C07288=1062.675,165.711,418.297,172.476,30.487,155.624
C07289=1062.681,165.960,418.274,172.478,30.490,155.624
C07290=1062.687,166.209,418.253,172.480,30.492,155.625
C07291=1062.693,166.458,418.230,172.483,30.496,155.625
C07292=1062.698,166.707,418.207,172.484,30.498,155.626
C07293=1062.704,166.956,418.185,172.486,30.501,155.626
C07294=1062.710,167.204,418.163,172.488,30.504,155.627
C07295=1062.715,167.454,418.140,172.490,30.507,155.627
C07296=1062.721,167.702,418.117,172.491,30.510,155.627
C07297=1062.727,167.952,418.096,172.494,30.513,155.628
C07298=1062.733,168.201,418.073,172.496,30.516,155.628
C07299=1062.738,168.449,418.050,172.498,30.519,155.629
C07300=1062.743,168.698,418.028,172.499,30.521,155.629
C07301=1062.750,168.947,418.006,172.501,30.524,155.630
C07302=1062.755,169.196,417.983,172.503,30.527,155.630
C07303=1062.761,169.445,417.960,172.506,30.530,155.631
C07304=1062.767,169.694,417.938,172.507,30.533,155.631
C07305=1062.773,169.943,417.916,172.509,30.536,155.632
C07306=1062.778,170.192,417.893,172.511,30.539,155.632
C07307=1062.784,170.440,417.870,172.513,30.541,155.632
C07308=1062.790,170.689,417.848,172.514,30.545,155.633
C07309=1062.795,170.939,417.826,172.517,30.547,155.633
C07310=1062.801,171.187,417.803,172.519,30.551,155.634
C07311=1062.807,171.436,417.780,172.521,30.553,155.634
C07312=1062.813,171.685,417.757,172.523,30.556,155.635
C07313=1062.819,171.934,417.735,172.524,30.559,155.635
C07314=1062.824,172.183,417.712,172.526,30.562,155.636
C07315=1062.830,172.431,417.690,172.529,30.565,155.636
C07316=1062.835,172.680,417.667,172.531,30.568,155.637
C07317=1062.842,172.930,417.645,172.532,30.571,155.637
C07318=1062.847,173.178,417.622,172.534,30.573,155.637
C07319=1062.853,173.427,417.599,172.536,30.576,155.638
C07320=1062.859,173.676,417.576,172.539,30.579,155.638
C07321=1062.865,173.925,417.554,172.540,30.582,155.639
C07322=1062.871,174.174,417.531,172.542,30.585,155.639
C07323=1062.877,174.458,417.506,172.545,30.589,155.640
C07324=1062.884,174.741,417.479,172.547,30.592,155.640
C07325=1062.891,175.024,417.453,172.549,30.595,155.641
C07326=1062.897,175.308,417.428,172.551,30.598,155.641
C07327=1062.903,175.557,417.405,172.553,30.601,155.642
C07328=1062.909,175.806,417.382,172.556,30.604,155.642
C07329=1062.914,176.055,417.359,172.557,30.607,155.643
C07330=1062.920,176.304,417.336,172.559,30.610,155.643
C07331=1062.927,176.552,417.314,172.561,30.612,155.644
C07332=1062.932,176.801,417.291,172.564,30.616,155.644
C07333=1062.938,177.050,417.268,172.565,30.618,155.645
C07334=1062.944,177.299,417.245,172.567,30.621,155.645
C07335=1062.950,177.548,417.222,172.569,30.624,155.646
C07336=1062.956,177.797,417.200,172.572,30.627,155.646
C07337=1062.962,178.045,417.177,172.573,30.630,155.646
C07338=1062.968,178.294,417.154,172.575,30.633,155.647
C07339=1062.974,178.544,417.131,172.577,30.636,155.647
C07340=1062.980,178.793,417.108,172.580,30.638,155.648
C07341=1062.985,179.042,417.085,172.581,30.642,155.648
C07342=1062.991,179.291,417.062,172.583,30.644,155.649
C07343=1062.997,179.539,417.039,172.585,30.647,155.649
C07344=1063.003,179.788,417.016,172.588,30.650,155.650
C07345=1063.009,180.037,416.993,172.590,30.653,155.650
C07346=1063.015,180.286,416.971,172.591,30.656,155.651
C07347=1063.020,180.535,416.948,172.593,30.659,155.651
C07348=1063.026,180.784,416.925,172.596,30.662,155.651
C07349=1063.033,181.033,416.901,172.598,30.665,155.652
C07350=1063.039,181.281,416.878,172.599,30.667,155.652
C07351=1063.045,181.530,416.855,172.601,30.670,155.653
C07352=1063.051,181.779,416.832,172.604,30.673,155.653
C07353=1063.056,182.028,416.809,172.606,30.676,155.654
C07354=1063.062,182.277,416.786,172.607,30.679,155.654
C07355=1063.068,182.526,416.764,172.610,30.682,155.655
C07356=1063.075,182.775,416.739,172.612,30.685,155.655
C07357=1063.080,183.024,416.717,172.614,30.687,155.655
C07358=1063.087,183.272,416.694,172.615,30.691,155.656
C07359=1063.092,183.521,416.671,172.618,30.693,155.656
C07360=1063.099,183.769,416.648,172.620,30.696,155.657
C07361=1063.105,184.019,416.624,172.622,30.699,155.657
C07362=1063.111,184.268,416.601,172.625,30.702,155.658
C07363=1063.116,184.517,416.578,172.626,30.705,155.658
C07364=1063.122,184.765,416.555,172.628,30.708,155.659
C07365=1063.127,185.014,416.531,172.631,30.711,155.659
C07366=1063.133,185.263,416.508,172.633,30.714,155.660
C07367=1063.139,185.511,416.485,172.634,30.717,155.660
C07368=1063.144,185.761,416.461,172.636,30.720,155.661
C07369=1063.150,186.010,416.438,172.639,30.723,155.661
C07370=1063.156,186.258,416.414,172.641,30.726,155.662
C07371=1063.161,186.508,416.391,172.642,30.730,155.662
C07372=1063.168,186.756,416.367,172.645,30.732,155.663
C07373=1063.172,187.005,416.343,172.647,30.736,155.663
C07374=1063.178,187.254,416.320,172.649,30.739,155.664
C07375=1063.184,187.502,416.297,172.650,30.742,155.664
C07376=1063.189,187.752,416.273,172.653,30.745,155.665
C07377=1063.195,188.000,416.250,172.655,30.748,155.665
C07378=1063.202,188.249,416.226,172.657,30.751,155.666
C07379=1063.207,188.498,416.202,172.659,30.754,155.666
C07380=1063.213,188.747,416.179,172.661,30.757,155.666
C07381=1063.218,188.996,416.155,172.663,30.760,155.667
C07382=1063.224,189.244,416.132,172.666,30.763,155.667
C07383=1063.230,189.493,416.108,172.668,30.766,155.668
C07384=1063.235,189.743,416.084,172.669,30.769,155.668
C07385=1063.241,189.991,416.061,172.672,30.773,155.669
C07386=1063.247,190.239,416.036,172.674,30.775,155.669
C07387=1063.253,190.523,416.010,172.677,30.779,155.670
C07388=1063.260,190.806,415.983,172.678,30.782,155.671
C07389=1063.267,191.089,415.957,172.681,30.786,155.671
C07390=1063.273,191.372,415.929,172.684,30.789,155.672
C07391=1063.279,191.620,415.906,172.686,30.792,155.672
C07392=1063.284,191.870,415.882,172.687,30.795,155.673
C07393=1063.290,192.118,415.858,172.690,30.798,155.673
C07394=1063.296,192.367,415.834,172.692,30.801,155.674
C07395=1063.301,192.616,415.811,172.694,30.805,155.674
C07396=1063.308,192.865,415.787,172.696,30.807,155.675
C07397=1063.313,193.114,415.762,172.698,30.811,155.675
C07398=1063.319,193.362,415.740,172.700,30.814,155.676
C07399=1063.325,193.612,415.715,172.703,30.817,155.676
C07400=1063.331,193.860,415.691,172.704,30.820,155.677
C07401=1063.336,194.109,415.668,172.707,30.823,155.677
C07402=1063.342,194.357,415.644,172.709,30.826,155.678
C07403=1063.348,194.607,415.619,172.711,30.829,155.678
C07404=1063.354,194.855,415.596,172.714,30.832,155.679
C07405=1063.359,195.104,415.572,172.715,30.835,155.679
C07406=1063.366,195.353,415.548,172.717,30.838,155.680
C07407=1063.372,195.601,415.525,172.720,30.842,155.680
C07408=1063.377,195.850,415.500,172.722,30.844,155.680
C07409=1063.384,196.099,415.476,172.724,30.848,155.681
C07410=1063.389,196.348,415.453,172.726,30.851,155.682
C07411=1063.395,196.597,415.429,172.728,30.853,155.682
C07412=1063.401,196.846,415.404,172.731,30.857,155.682
C07413=1063.407,197.094,415.381,172.732,30.860,155.683
C07414=1063.412,197.343,415.357,172.735,30.863,155.683
C07415=1063.419,197.592,415.332,172.737,30.866,155.684
C07416=1063.424,197.840,415.308,172.739,30.869,155.684
C07417=1063.430,198.089,415.284,172.742,30.872,155.685
C07418=1063.435,198.338,415.261,172.743,30.875,155.685
C07419=1063.441,198.587,415.237,172.746,30.879,155.686
C07420=1063.447,198.836,415.212,172.748,30.881,155.686
C07421=1063.453,199.084,415.189,172.751,30.884,155.687
C07422=1063.459,199.334,415.164,172.752,30.888,155.687
C07423=1063.465,199.582,415.140,172.754,30.891,155.688
C07424=1063.471,199.831,415.116,172.757,30.894,155.688
C07425=1063.477,200.079,415.092,172.759,30.897,155.689
C07426=1063.483,200.328,415.068,172.761,30.900,155.689
C07427=1063.489,200.577,415.044,172.763,30.903,155.690
C07428=1063.495,200.826,415.020,172.766,30.906,155.690
C07429=1063.500,201.075,414.995,172.768,30.909,155.691
C07430=1063.506,201.323,414.971,172.770,30.912,155.691
C07431=1063.512,201.572,414.947,172.772,30.915,155.692
C07432=1063.518,201.821,414.923,172.774,30.919,155.692
C07433=1063.524,202.070,414.898,172.777,30.921,155.693
C07434=1063.530,202.318,414.875,172.779,30.925,155.693
C07435=1063.537,202.567,414.849,172.781,30.928,155.694
C07436=1063.542,202.816,414.825,172.783,30.931,155.694
C07437=1063.548,203.065,414.801,172.786,30.934,155.695
C07438=1063.553,203.313,414.776,172.788,30.938,155.695
C07439=1063.559,203.562,414.753,172.790,30.941,155.696
C07440=1063.565,203.811,414.728,172.792,30.944,155.697
C07441=1063.571,204.059,414.703,172.794,30.947,155.697
C07442=1063.576,204.308,414.678,172.797,30.950,155.697
C07443=1063.582,204.557,414.654,172.799,30.953,155.698
C07444=1063.588,204.806,414.630,172.801,30.957,155.699
C07445=1063.594,205.054,414.606,172.803,30.960,155.699
C07446=1063.600,205.303,414.581,172.806,30.963,155.700
C07447=1063.605,205.552,414.556,172.808,30.966,155.700
C07448=1063.611,205.801,414.532,172.811,30.970,155.701
C07449=1063.617,206.049,414.507,172.812,30.973,155.701
C07450=1063.623,206.298,414.482,172.815,30.976,155.702
C07451=1063.647,207.346,414.379,172.981,31.057,155.708
C07452=1063.653,207.569,414.356,172.982,31.060,155.709
C07453=1063.659,207.793,414.333,172.984,31.064,155.710
C07454=1063.664,208.016,414.311,172.986,31.068,155.710
C07455=1063.669,208.240,414.288,172.988,31.071,155.711
C07456=1063.675,208.463,414.265,172.988,31.075,155.712
C07457=1063.680,208.688,414.242,172.990,31.079,155.712
C07458=1063.685,208.910,414.219,172.992,31.082,155.713
C07459=1063.691,209.134,414.196,172.994,31.086,155.714
C07460=1063.697,209.383,414.171,172.996,31.090,155.714
C07461=1063.703,209.631,414.146,172.998,31.094,155.715
C07462=1063.709,209.880,414.120,173.000,31.098,155.716
C07463=1063.715,210.129,414.094,173.002,31.102,155.717
C07464=1063.721,210.378,414.069,173.004,31.106,155.717
C07465=1063.728,210.626,414.043,173.006,31.111,155.718
C07466=1063.733,210.875,414.017,173.008,31.114,155.719
C07467=1063.739,211.123,413.992,173.010,31.119,155.720
C07468=1063.745,211.372,413.966,173.012,31.122,155.720
C07469=1063.752,211.621,413.941,173.014,31.127,155.721
C07470=1063.757,211.869,413.915,173.016,31.131,155.722
C07471=1063.763,212.117,413.889,173.018,31.135,155.722
C07472=1063.769,212.366,413.864,173.020,31.139,155.723
C07473=1063.775,212.615,413.838,173.022,31.143,155.724
C07474=1063.781,212.863,413.813,173.024,31.147,155.725
C07475=1063.787,213.112,413.787,173.026,31.151,155.725
C07476=1063.793,213.360,413.761,173.027,31.155,155.726
C07477=1063.799,213.609,413.735,173.030,31.159,155.727
C07478=1063.805,213.858,413.710,173.032,31.164,155.728
C07479=1063.811,214.106,413.683,173.034,31.167,155.728
C07480=1063.817,214.355,413.658,173.036,31.172,155.729
C07481=1063.823,214.604,413.632,173.037,31.175,155.730
C07482=1063.829,214.852,413.607,173.040,31.180,155.730
C07483=1063.835,215.101,413.580,173.042,31.184,155.731
C07484=1063.841,215.349,413.555,173.044,31.188,155.732
C07485=1063.847,215.598,413.528,173.045,31.192,155.733
C07486=1063.853,215.846,413.503,173.048,31.196,155.733
C07487=1063.858,216.095,413.477,173.050,31.200,155.734
C07488=1063.865,216.343,413.451,173.052,31.204,155.735
C07489=1063.871,216.592,413.426,173.054,31.208,155.736
C07490=1063.877,216.840,413.399,173.056,31.212,155.736
C07491=1063.884,217.090,413.373,173.058,31.216,155.737
C07492=1063.889,217.339,413.347,173.060,31.220,155.738
C07493=1063.896,217.587,413.321,173.062,31.225,155.738
C07494=1063.901,217.836,413.295,173.064,31.228,155.739
C07495=1063.908,218.084,413.269,173.066,31.233,155.740
C07496=1063.913,218.333,413.243,173.068,31.236,155.741
C07497=1063.920,218.581,413.217,173.070,31.240,155.741
C07498=1063.925,218.830,413.191,173.072,31.244,155.742
C07499=1063.932,219.078,413.165,173.074,31.248,155.743
C07500=1063.937,219.327,413.139,173.077,31.253,155.743
C07501=1063.944,219.576,413.113,173.079,31.256,155.744
C07502=1063.950,219.825,413.087,173.080,31.261,155.745
C07503=1063.956,220.073,413.061,173.083,31.264,155.746
C07504=1063.962,220.321,413.034,173.085,31.268,155.746
C07505=1063.968,220.570,413.009,173.087,31.272,155.747
C07506=1063.974,220.818,412.982,173.088,31.276,155.748
C07507=1063.980,221.067,412.957,173.091,31.281,155.748
C07508=1063.985,221.293,412.933,173.093,31.284,155.749
C07509=1063.991,221.519,412.909,173.095,31.287,155.750
C07510=1063.996,221.745,412.885,173.097,31.291,155.750
C07511=1064.002,221.971,412.861,173.098,31.295,155.751
C07512=1064.008,222.197,412.837,173.100,31.299,155.752
C07513=1064.013,222.423,412.813,173.102,31.302,155.752
C07514=1064.019,222.649,412.789,173.104,31.306,155.753
C07515=1064.023,222.875,412.765,173.106,31.310,155.754
C07516=1064.030,223.124,412.738,173.108,31.314,155.754
C07517=1064.036,223.372,412.712,173.110,31.318,155.755
C07518=1064.042,223.621,412.686,173.112,31.322,155.756
C07519=1064.047,223.869,412.660,173.115,31.326,155.757
C07520=1064.053,224.118,412.633,173.116,31.330,155.757
C07521=1064.060,224.366,412.607,173.118,31.334,155.758
C07522=1064.066,224.615,412.580,173.121,31.338,155.759
C07523=1064.072,224.864,412.554,173.123,31.342,155.759
C07524=1064.077,225.112,412.527,173.125,31.346,155.760
C07525=1064.084,225.360,412.501,173.127,31.350,155.761
C07526=1064.090,225.608,412.475,173.129,31.354,155.762
C07527=1064.096,225.857,412.448,173.131,31.358,155.762
C07528=1064.102,226.106,412.421,173.134,31.362,155.763
C07529=1064.107,226.355,412.395,173.135,31.366,155.764
C07530=1064.114,226.603,412.369,173.137,31.370,155.764
C07531=1064.120,226.852,412.342,173.140,31.374,155.765
C07532=1064.126,227.100,412.315,173.142,31.378,155.766
C07533=1064.132,227.349,412.289,173.145,31.382,155.767
C07534=1064.137,227.597,412.262,173.146,31.386,155.767
C07535=1064.145,227.846,412.236,173.148,31.390,155.768
C07536=1064.150,228.094,412.209,173.151,31.394,155.769
C07537=1064.156,228.342,412.182,173.153,31.398,155.769
C07538=1064.163,228.592,412.155,173.154,31.402,155.770
C07539=1064.168,228.840,412.129,173.157,31.406,155.771
C07540=1064.175,229.088,412.102,173.159,31.409,155.772
C07541=1064.181,229.337,412.075,173.161,31.414,155.772
C07542=1064.187,229.585,412.049,173.164,31.417,155.773
C07543=1064.193,229.834,412.022,173.165,31.422,155.774
C07544=1064.199,230.083,411.995,173.168,31.426,155.774
C07545=1064.205,230.331,411.969,173.170,31.429,155.775
C07546=1064.211,230.580,411.942,173.172,31.434,155.776
C07547=1064.216,230.828,411.915,173.175,31.437,155.777
C07548=1064.223,231.076,411.887,173.176,31.442,155.777
C07549=1064.229,231.325,411.861,173.179,31.445,155.778
C07550=1064.235,231.573,411.834,173.181,31.450,155.779
C07551=1064.241,231.822,411.807,173.183,31.453,155.779
C07552=1064.247,232.070,411.781,173.186,31.457,155.780
C07553=1064.253,232.319,411.754,173.187,31.462,155.781
C07554=1064.259,232.567,411.726,173.189,31.465,155.782
C07555=1064.265,232.816,411.700,173.192,31.470,155.782
C07556=1064.271,233.064,411.673,173.194,31.473,155.783
C07557=1064.277,233.313,411.646,173.197,31.477,155.784
C07558=1064.283,233.561,411.619,173.198,31.481,155.784
C07559=1064.289,233.810,411.591,173.200,31.485,155.785
C07560=1064.295,234.059,411.564,173.203,31.490,155.786
C07561=1064.300,234.307,411.538,173.205,31.493,155.787
C07562=1064.307,234.555,411.510,173.208,31.498,155.787
C07563=1064.313,234.804,411.483,173.209,31.501,155.788
C07564=1064.318,235.026,411.459,173.211,31.505,155.789
C07565=1064.323,235.248,411.435,173.213,31.508,155.789
C07566=1064.329,235.470,411.410,173.216,31.512,155.790
C07567=1064.334,235.691,411.386,173.218,31.516,155.791
C07568=1064.340,235.914,411.362,173.219,31.519,155.791
C07569=1064.345,236.136,411.337,173.221,31.523,155.792
C07570=1064.351,236.358,411.313,173.223,31.526,155.792
C07571=1064.356,236.580,411.289,173.225,31.530,155.793
C07572=1064.361,236.828,411.262,173.228,31.534,155.794
C07573=1064.368,237.077,411.235,173.230,31.538,155.795
C07574=1064.374,237.325,411.207,173.232,31.542,155.795
C07575=1064.380,237.574,411.180,173.234,31.545,155.796
C07576=1064.386,237.822,411.153,173.237,31.550,155.797
C07577=1064.392,238.071,411.126,173.239,31.554,155.797
C07578=1064.398,238.319,411.098,173.242,31.557,155.798
C07579=1064.404,238.568,411.071,173.243,31.562,155.799
C07580=1064.410,238.816,411.044,173.245,31.565,155.800
C07581=1064.416,239.065,411.016,173.248,31.569,155.800
C07582=1064.422,239.313,410.989,173.250,31.573,155.801
C07583=1064.429,239.562,410.962,173.253,31.577,155.802
C07584=1064.435,239.809,410.934,173.254,31.581,155.802
C07585=1064.441,240.058,410.906,173.257,31.585,155.803
C07586=1064.446,240.307,410.879,173.259,31.589,155.804
C07587=1064.453,240.555,410.852,173.262,31.593,155.805
C07588=1064.458,240.804,410.824,173.264,31.597,155.805
C07589=1064.465,241.052,410.797,173.267,31.601,155.806
C07590=1064.471,241.300,410.769,173.268,31.605,155.807
C07591=1064.477,241.549,410.742,173.271,31.609,155.807
C07592=1064.483,241.797,410.714,173.273,31.613,155.808
C07593=1064.489,242.045,410.687,173.276,31.617,155.809
C07594=1064.495,242.294,410.660,173.278,31.621,155.809
C07595=1064.501,242.542,410.632,173.280,31.625,155.810
C07596=1064.508,242.791,410.604,173.282,31.629,155.811
C07597=1064.513,243.040,410.577,173.284,31.632,155.812
C07598=1064.519,243.288,410.549,173.287,31.636,155.812
C07599=1064.525,243.536,410.521,173.289,31.641,155.813
C07600=1064.531,243.785,410.493,173.292,31.644,155.814
C07601=1064.537,244.033,410.465,173.293,31.649,155.815
C07602=1064.543,244.282,410.438,173.296,31.652,155.815
C07603=1064.548,244.530,410.410,173.298,31.657,155.816
C07604=1064.555,244.778,410.383,173.301,31.660,155.817
C07605=1064.560,245.026,410.355,173.303,31.664,155.817
C07606=1064.567,245.275,410.327,173.305,31.669,155.818
C07607=1064.573,245.523,410.299,173.307,31.672,155.819
C07608=1064.579,245.771,410.271,173.310,31.676,155.819
C07609=1064.585,246.021,410.244,173.312,31.680,155.820
C07610=1064.591,246.268,410.216,173.315,31.684,155.821
C07611=1064.597,246.517,410.188,173.317,31.688,155.822
C07612=1064.603,246.766,410.160,173.319,31.692,155.822
C07613=1064.609,247.013,410.132,173.322,31.696,155.823
C07614=1064.615,247.262,410.104,173.324,31.700,155.824
C07615=1064.620,247.510,410.076,173.327,31.704,155.824
C07616=1064.626,247.759,410.048,173.329,31.708,155.825
C07617=1064.633,248.007,410.020,173.332,31.712,155.826
C07618=1064.638,248.256,409.992,173.333,31.716,155.827
C07619=1064.644,248.504,409.964,173.336,31.720,155.827
C07620=1064.649,248.723,409.939,173.338,31.724,155.828
C07621=1064.654,248.942,409.914,173.340,31.727,155.829
C07622=1064.660,249.161,409.889,173.342,31.731,155.829
C07623=1064.665,249.380,409.864,173.345,31.734,155.830
C07624=1064.670,249.599,409.840,173.346,31.738,155.831
C07625=1064.675,249.818,409.815,173.348,31.741,155.831
C07626=1064.681,250.036,409.790,173.350,31.745,155.832
C07627=1064.686,250.255,409.765,173.352,31.748,155.833
C07628=1064.692,250.502,409.737,173.355,31.752,155.833
C07629=1064.698,250.751,409.709,173.358,31.757,155.834
C07630=1064.704,251.000,409.681,173.360,31.760,155.835
C07631=1064.709,251.248,409.653,173.362,31.764,155.835
C07632=1064.715,251.497,409.624,173.364,31.768,155.836
C07633=1064.722,251.745,409.597,173.367,31.772,155.837
C07634=1064.728,251.993,409.568,173.369,31.776,155.838
C07635=1064.734,252.241,409.540,173.372,31.780,155.838
C07636=1064.739,252.490,409.511,173.375,31.784,155.839
C07637=1064.745,252.739,409.483,173.376,31.788,155.840
C07638=1064.752,252.986,409.455,173.379,31.792,155.840
C07639=1064.758,253.235,409.427,173.381,31.796,155.841
C07640=1064.764,253.483,409.398,173.384,31.800,155.842
C07641=1064.770,253.732,409.369,173.386,31.804,155.843
C07642=1064.775,253.980,409.341,173.389,31.808,155.843
C07643=1064.782,254.228,409.313,173.391,31.812,155.844
C07644=1064.788,254.476,409.284,173.393,31.816,155.845
C07645=1064.794,254.725,409.256,173.396,31.820,155.845
C07646=1064.800,254.973,409.228,173.398,31.823,155.846
C07647=1064.806,255.221,409.199,173.401,31.828,155.847
C07648=1064.812,255.470,409.171,173.404,31.832,155.848
C07649=1064.819,255.718,409.142,173.406,31.835,155.848
C07650=1064.825,255.966,409.114,173.408,31.840,155.849
C07651=1064.830,256.214,409.085,173.410,31.843,155.850
C07652=1064.836,256.463,409.057,173.413,31.847,155.850
C07653=1064.842,256.711,409.029,173.416,31.851,155.851
C07654=1064.848,256.960,409.000,173.418,31.855,155.852
C07655=1064.854,257.208,408.971,173.421,31.859,155.853
C07656=1064.861,257.456,408.943,173.422,31.863,155.853
C07657=1064.867,257.705,408.915,173.425,31.867,155.854
C07658=1064.873,257.952,408.886,173.428,31.871,155.855
C07659=1064.879,258.200,408.857,173.430,31.875,155.855
C07660=1064.885,258.449,408.829,173.433,31.879,155.856
C07661=1064.891,258.697,408.799,173.436,31.883,155.857
C07662=1064.897,258.946,408.771,173.438,31.887,155.858
C07663=1064.904,259.194,408.742,173.440,31.891,155.858
C07664=1064.910,259.443,408.714,173.443,31.894,155.859
C07665=1064.917,259.691,408.685,173.445,31.898,155.860
C07666=1064.923,259.939,408.656,173.448,31.902,155.860
C07667=1064.929,260.188,408.628,173.450,31.906,155.861
C07668=1064.935,260.436,408.599,173.453,31.910,155.862
C07669=1064.941,260.684,408.570,173.456,31.914,155.863
C07670=1064.947,260.932,408.542,173.457,31.918,155.863
C07671=1064.953,261.180,408.513,173.460,31.922,155.864
C07672=1064.959,261.428,408.484,173.463,31.926,155.865
C07673=1064.965,261.676,408.455,173.465,31.929,155.865
C07674=1064.971,261.925,408.426,173.468,31.933,155.866
C07675=1064.977,262.173,408.397,173.471,31.938,155.867
C07676=1064.984,262.391,408.373,173.473,31.941,155.867
C07677=1064.989,262.609,408.347,173.475,31.944,155.868
C07678=1064.994,262.827,408.322,173.477,31.948,155.869
C07679=1065.000,263.045,408.296,173.479,31.951,155.869
C07680=1065.006,263.262,408.271,173.482,31.954,155.870
C07681=1065.011,263.480,408.246,173.484,31.958,155.871
C07682=1065.016,263.698,408.220,173.486,31.961,155.871
C07683=1065.022,263.915,408.194,173.489,31.965,155.872
C07684=1065.028,264.164,408.166,173.491,31.969,155.872
C07685=1065.033,264.412,408.136,173.493,31.973,155.873
C07686=1065.040,264.661,408.107,173.496,31.977,155.874
C07687=1065.045,264.908,408.079,173.498,31.981,155.875
C07688=1065.052,265.156,408.050,173.501,31.985,155.875
C07689=1065.057,265.405,408.020,173.504,31.989,155.876
C07690=1065.063,265.653,407.991,173.506,31.993,155.877
C07691=1065.070,265.901,407.962,173.509,31.996,155.878
C07692=1065.076,266.149,407.933,173.511,32.001,155.878
C07693=1065.081,266.397,407.903,173.514,32.005,155.879
C07694=1065.088,266.645,407.874,173.516,32.009,155.880
C07695=1065.094,266.894,407.845,173.519,32.012,155.880
C07696=1065.100,267.143,407.815,173.522,32.017,155.881
C07697=1065.106,267.391,407.786,173.524,32.020,155.882
C07698=1065.112,267.639,407.757,173.527,32.024,155.883
C07699=1065.119,267.887,407.727,173.530,32.029,155.883
C07700=1065.125,268.135,407.698,173.531,32.032,155.884
C07701=1065.131,268.383,407.669,173.534,32.037,155.885
C07702=1065.137,268.631,407.640,173.537,32.040,155.886
C07703=1065.143,268.880,407.610,173.540,32.044,155.886
C07704=1065.149,269.128,407.581,173.542,32.048,155.887
C07705=1065.155,269.376,407.552,173.545,32.052,155.888
C07706=1065.161,269.624,407.521,173.548,32.056,155.888
C07707=1065.167,269.872,407.492,173.551,32.060,155.889
C07708=1065.173,270.120,407.463,173.552,32.064,155.890
C07709=1065.179,270.369,407.433,173.555,32.068,155.891
C07710=1065.185,270.617,407.403,173.558,32.072,155.891
C07711=1065.192,270.865,407.374,173.561,32.076,155.892
C07712=1065.198,271.113,407.345,173.563,32.080,155.893
C07713=1065.203,271.362,407.315,173.566,32.084,155.894
C07714=1065.210,271.609,407.286,173.569,32.088,155.894
C07715=1065.215,271.858,407.256,173.572,32.092,155.895
C07716=1065.222,272.105,407.226,173.573,32.096,155.896
C07717=1065.228,272.354,407.196,173.576,32.100,155.897
C07718=1065.234,272.602,407.167,173.579,32.104,155.897
C07719=1065.240,272.850,407.137,173.582,32.108,155.898
C07720=1065.246,273.098,407.108,173.584,32.112,155.899
C07721=1065.252,273.347,407.078,173.587,32.116,155.899
C07722=1065.258,273.594,407.048,173.590,32.120,155.900
C07723=1065.264,273.843,407.019,173.593,32.124,155.901
C07724=1065.271,274.091,406.989,173.594,32.128,155.902
C07725=1065.277,274.339,406.959,173.597,32.132,155.902
C07726=1065.282,274.587,406.929,173.600,32.136,155.903
C07727=1065.289,274.835,406.900,173.603,32.140,155.904
C07728=1065.294,275.083,406.869,173.606,32.144,155.905
C07729=1065.301,275.332,406.840,173.608,32.148,155.905
C07730=1065.307,275.580,406.809,173.611,32.152,155.906
C07731=1065.313,275.828,406.779,173.614,32.156,155.907
C07732=1065.318,276.048,406.753,173.616,32.160,155.908
C07733=1065.323,276.267,406.727,173.618,32.163,155.908
C07734=1065.329,276.487,406.700,173.620,32.167,155.909
C07735=1065.335,276.706,406.674,173.623,32.170,155.909
C07736=1065.340,276.925,406.647,173.625,32.174,155.910
C07737=1065.346,277.145,406.621,173.628,32.178,155.911
C07738=1065.350,277.364,406.594,173.630,32.181,155.911
C07739=1065.356,277.584,406.567,173.633,32.185,155.912
C07740=1065.362,277.832,406.538,173.636,32.189,155.913
C07741=1065.368,278.080,406.507,173.638,32.192,155.914
C07742=1065.374,278.328,406.477,173.641,32.197,155.914
C07743=1065.380,278.577,406.447,173.643,32.201,155.915
C07744=1065.387,278.825,406.417,173.646,32.205,155.916
C07745=1065.393,279.073,406.387,173.649,32.209,155.916
C07746=1065.399,279.321,406.356,173.651,32.213,155.917
C07747=1065.405,279.569,406.327,173.654,32.217,155.918
C07748=1065.411,279.817,406.297,173.657,32.221,155.919
C07749=1065.417,280.066,406.266,173.660,32.225,155.920
C07750=1065.423,280.313,406.236,173.663,32.229,155.920
C07751=1065.429,280.561,406.205,173.666,32.233,155.921
C07752=1065.436,280.809,406.176,173.667,32.237,155.922
C07753=1065.442,281.058,406.146,173.670,32.241,155.923
C07754=1065.448,281.306,406.115,173.673,32.245,155.923
C07755=1065.453,281.553,406.085,173.676,32.249,155.924
C07756=1065.460,281.802,406.054,173.679,32.253,155.925
C07757=1065.466,282.050,406.024,173.682,32.258,155.926
C07758=1065.471,282.298,405.993,173.684,32.261,155.926
C07759=1065.478,282.546,405.963,173.687,32.266,155.927
C07760=1065.484,282.794,405.932,173.690,32.269,155.928
C07761=1065.489,283.042,405.902,173.693,32.274,155.929
C07762=1065.496,283.290,405.871,173.695,32.278,155.929
C07763=1065.502,283.538,405.841,173.698,32.282,155.930
C07764=1065.508,283.786,405.811,173.701,32.286,155.931
C07765=1065.514,284.034,405.780,173.704,32.290,155.932
C07766=1065.520,284.282,405.750,173.706,32.294,155.932
C07767=1065.526,284.531,405.719,173.709,32.298,155.933
C07768=1065.532,284.778,405.688,173.712,32.302,155.934
C07769=1065.539,285.026,405.658,173.715,32.306,155.935
C07770=1065.545,285.274,405.627,173.718,32.310,155.935
C07771=1065.551,285.522,405.597,173.721,32.314,155.936
C07772=1065.558,285.770,405.566,173.724,32.318,155.937
C07773=1065.563,286.018,405.536,173.726,32.323,155.938
C07774=1065.570,286.266,405.504,173.728,32.326,155.938
C07775=1065.576,286.514,405.474,173.731,32.331,155.939
C07776=1065.582,286.762,405.444,173.734,32.335,155.940
C07777=1065.588,287.010,405.413,173.737,32.339,155.941
C07778=1065.594,287.258,405.383,173.740,32.343,155.941
C07779=1065.601,287.506,405.351,173.743,32.347,155.942
C07780=1065.606,287.754,405.321,173.746,32.351,155.943
C07781=1065.613,288.002,405.290,173.749,32.355,155.944
C07782=1065.619,288.250,405.259,173.752,32.359,155.945
C07783=1065.625,288.498,405.228,173.755,32.363,155.945
C07784=1065.631,288.746,405.197,173.757,32.367,155.946
C07785=1065.637,288.994,405.166,173.760,32.372,155.947
C07786=1065.643,289.242,405.136,173.762,32.375,155.947
C07787=1065.649,289.490,405.105,173.765,32.380,155.948
C07788=1065.654,289.715,405.077,173.768,32.383,155.949
C07789=1065.661,289.940,405.049,173.771,32.387,155.950
C07790=1065.666,290.165,405.020,173.773,32.391,155.950
C07791=1065.672,290.389,404.993,173.776,32.394,155.951
C07792=1065.677,290.614,404.964,173.779,32.399,155.952
C07793=1065.683,290.839,404.936,173.781,32.402,155.953
C07794=1065.688,291.063,404.908,173.784,32.406,155.953
C07795=1065.694,291.288,404.879,173.787,32.410,155.954
C07796=1065.700,291.536,404.849,173.789,32.414,155.955
C07797=1065.706,291.784,404.818,173.792,32.418,155.955
C07798=1065.712,292.032,404.787,173.795,32.422,155.956
C07799=1065.718,292.280,404.755,173.798,32.426,155.957
C07800=1065.725,292.529,404.724,173.801,32.430,155.958
C07801=1065.731,292.776,404.693,173.803,32.435,155.959
C07802=1065.737,293.024,404.661,173.806,32.438,155.959
C07803=1065.743,293.272,404.631,173.809,32.443,155.960
C07804=1065.749,293.520,404.600,173.812,32.447,155.961
C07805=1065.755,293.768,404.568,173.815,32.451,155.962
C07806=1065.761,294.016,404.537,173.818,32.455,155.962
C07807=1065.768,294.264,404.506,173.821,32.459,155.963
C07808=1065.774,294.511,404.475,173.824,32.463,155.964
C07809=1065.780,294.760,404.443,173.827,32.468,155.965
C07810=1065.786,295.008,404.412,173.829,32.472,155.966
C07811=1065.792,295.255,404.380,173.832,32.476,155.966
C07812=1065.799,295.503,404.349,173.835,32.480,155.967
C07813=1065.805,295.752,404.318,173.838,32.484,155.968
C07814=1065.810,295.999,404.286,173.841,32.488,155.969
C07815=1065.817,296.247,404.255,173.844,32.493,155.969
C07816=1065.823,296.495,404.223,173.847,32.497,155.970
C07817=1065.829,296.742,404.192,173.850,32.501,155.971
C07818=1065.835,296.991,404.160,173.853,32.505,155.972
C07819=1065.842,297.239,404.129,173.856,32.510,155.973
C07820=1065.847,297.487,404.098,173.859,32.514,155.974
C07821=1065.854,297.735,404.066,173.862,32.518,155.974
C07822=1065.860,297.983,404.034,173.865,32.522,155.975
C07823=1065.865,298.230,404.002,173.868,32.527,155.976
C07824=1065.872,298.478,403.971,173.871,32.531,155.977
C07825=1065.878,298.726,403.939,173.873,32.535,155.978
C07826=1065.883,298.974,403.907,173.876,32.539,155.978
C07827=1065.889,299.222,403.875,173.879,32.544,155.979
C07828=1065.896,299.470,403.844,173.882,32.548,155.980
C07829=1065.902,299.717,403.811,173.885,32.552,155.981
C07830=1065.908,299.965,403.779,173.888,32.556,155.982
C07831=1065.914,300.213,403.748,173.891,32.561,155.982
C07832=1065.920,300.461,403.716,173.895,32.565,155.983
C07833=1065.926,300.709,403.684,173.898,32.569,155.984
C07834=1065.932,300.957,403.652,173.901,32.574,155.985
C07835=1065.938,301.205,403.621,173.904,32.578,155.986
C07836=1065.944,301.452,403.589,173.907,32.583,155.987
C07837=1065.950,301.700,403.556,173.910,32.587,155.987
C07838=1065.956,301.948,403.524,173.913,32.591,155.988
C07839=1065.963,302.196,403.493,173.916,32.595,155.989
C07840=1065.968,302.444,403.461,173.919,32.600,155.990
C07841=1065.974,302.691,403.429,173.922,32.604,155.991
C07842=1065.980,302.939,403.397,173.924,32.608,155.991
C07843=1065.987,303.187,403.365,173.927,32.612,155.992
C07844=1065.993,303.419,403.335,173.930,32.617,155.993
C07845=1065.998,303.651,403.305,173.933,32.620,155.994
C07846=1066.004,303.884,403.275,173.936,32.624,155.994
C07847=1066.010,304.116,403.245,173.939,32.629,155.995
C07848=1066.016,304.349,403.214,173.942,32.632,155.996
C07849=1066.021,304.581,403.185,173.945,32.637,155.997
C07850=1066.027,304.813,403.155,173.947,32.641,155.998
C07851=1066.033,305.045,403.125,173.950,32.644,155.998
C07852=1066.039,305.293,403.092,173.953,32.649,155.999
C07853=1066.045,305.541,403.060,173.957,32.654,156.000
C07854=1066.051,305.789,403.027,173.960,32.658,156.001
C07855=1066.058,306.037,402.996,173.963,32.662,156.002
C07856=1066.064,306.284,402.963,173.966,32.666,156.002
C07857=1066.070,306.533,402.931,173.969,32.670,156.003
C07858=1066.076,306.779,402.899,173.972,32.675,156.004
C07859=1066.082,307.028,402.867,173.975,32.679,156.005
C07860=1066.089,307.275,402.834,173.978,32.683,156.006
C07861=1066.095,307.523,402.802,173.982,32.688,156.007
C07862=1066.101,307.771,402.770,173.985,32.692,156.007
C07863=1066.107,308.019,402.738,173.988,32.697,156.008
C07864=1066.114,308.267,402.705,173.990,32.701,156.009
C07865=1066.120,308.514,402.672,173.993,32.705,156.010
C07866=1066.127,308.762,402.641,173.996,32.709,156.011
C07867=1066.133,309.010,402.608,173.999,32.713,156.011
C07868=1066.139,309.258,402.576,174.003,32.718,156.012
C07869=1066.145,309.505,402.543,174.006,32.723,156.013
C07870=1066.151,309.753,402.511,174.009,32.727,156.014
C07871=1066.158,310.001,402.478,174.012,32.731,156.015
C07872=1066.164,310.249,402.446,174.015,32.735,156.016
C07873=1066.170,310.496,402.413,174.018,32.740,156.017
C07874=1066.177,310.744,402.381,174.022,32.744,156.017
C07875=1066.184,310.992,402.348,174.025,32.749,156.018
C07876=1066.190,311.240,402.316,174.028,32.753,156.019
C07877=1066.196,311.488,402.283,174.031,32.757,156.020
C07878=1066.203,311.735,402.250,174.034,32.761,156.021
C07879=1066.209,311.983,402.217,174.038,32.766,156.022
C07880=1066.215,312.231,402.185,174.041,32.770,156.022
C07881=1066.221,312.479,402.153,174.044,32.775,156.023
C07882=1066.227,312.726,402.120,174.047,32.779,156.024
C07883=1066.234,312.975,402.087,174.050,32.783,156.025
C07884=1066.241,313.222,402.054,174.054,32.788,156.026
C07885=1066.247,313.470,402.021,174.057,32.792,156.027
C07886=1066.254,313.717,401.989,174.060,32.796,156.027
C07887=1066.260,313.965,401.956,174.063,32.800,156.028
C07888=1066.266,314.213,401.923,174.066,32.805,156.029
C07889=1066.272,314.460,401.890,174.070,32.810,156.030
C07890=1066.278,314.708,401.858,174.073,32.814,156.031
C07891=1066.284,314.956,401.824,174.076,32.819,156.032
C07892=1066.291,315.204,401.791,174.079,32.823,156.033
C07893=1066.296,315.452,401.758,174.082,32.828,156.034
C07894=1066.303,315.700,401.725,174.086,32.832,156.034
C07895=1066.309,315.947,401.692,174.089,32.837,156.035
C07896=1066.315,316.194,401.658,174.092,32.841,156.036
C07897=1066.321,316.442,401.626,174.095,32.846,156.037
C07898=1066.327,316.690,401.592,174.098,32.851,156.038
C07899=1066.333,316.938,401.560,174.102,32.855,156.039
C07900=1066.339,317.171,401.528,174.105,32.859,156.040
C07901=1066.345,317.406,401.496,174.108,32.864,156.041
C07902=1066.350,317.640,401.465,174.111,32.868,156.041
C07903=1066.357,317.874,401.433,174.114,32.872,156.042
C07904=1066.362,318.109,401.402,174.117,32.877,156.043
C07905=1066.368,318.342,401.371,174.120,32.881,156.044
C07906=1066.374,318.576,401.339,174.123,32.886,156.045
C07907=1066.380,318.811,401.307,174.126,32.890,156.046
C07908=1066.386,319.058,401.274,174.128,32.894,156.046
C07909=1066.392,319.306,401.241,174.132,32.899,156.047
C07910=1066.398,319.554,401.208,174.135,32.904,156.048
C07911=1066.405,319.802,401.174,174.138,32.908,156.049
C07912=1066.411,320.049,401.141,174.141,32.913,156.050
C07913=1066.417,320.297,401.107,174.145,32.917,156.051
C07914=1066.423,320.544,401.074,174.148,32.922,156.052
C07915=1066.429,320.793,401.040,174.151,32.926,156.053
C07916=1066.436,321.040,401.007,174.154,32.931,156.054
C07917=1066.441,321.288,400.973,174.158,32.935,156.054
C07918=1066.448,321.535,400.940,174.161,32.940,156.055
C07919=1066.454,321.783,400.906,174.164,32.945,156.056
C07920=1066.461,322.030,400.873,174.168,32.949,156.057
C07921=1066.467,322.279,400.839,174.171,32.954,156.058
C07922=1066.473,322.526,400.806,174.174,32.959,156.059
C07923=1066.479,322.773,400.772,174.177,32.963,156.060
C07924=1066.486,323.021,400.739,174.181,32.968,156.061
C07925=1066.492,323.269,400.704,174.185,32.972,156.062
C07926=1066.498,323.516,400.672,174.188,32.977,156.063
C07927=1066.505,323.764,400.637,174.192,32.982,156.064
C07928=1066.511,324.011,400.604,174.195,32.986,156.064
C07929=1066.518,324.260,400.570,174.198,32.991,156.065
C07930=1066.523,324.507,400.536,174.202,32.996,156.066
C07931=1066.531,324.755,400.502,174.205,33.000,156.067
C07932=1066.536,325.003,400.469,174.208,33.005,156.068
C07933=1066.543,325.250,400.435,174.212,33.009,156.069
C07934=1066.549,325.498,400.401,174.215,33.014,156.070
C07935=1066.556,325.745,400.368,174.218,33.019,156.071
C07936=1066.562,325.993,400.333,174.222,33.024,156.072
C07937=1066.568,326.240,400.300,174.225,33.028,156.073
C07938=1066.575,326.488,400.266,174.228,33.033,156.074
C07939=1066.581,326.736,400.232,174.232,33.037,156.075
C07940=1066.588,326.983,400.198,174.235,33.042,156.075
C07941=1066.595,327.231,400.164,174.238,33.047,156.076
C07942=1066.600,327.478,400.130,174.242,33.052,156.077
C07943=1066.608,327.726,400.096,174.245,33.056,156.078
C07944=1066.613,327.974,400.062,174.249,33.061,156.079
C07945=1066.620,328.222,400.029,174.252,33.065,156.080
C07946=1066.626,328.469,399.995,174.255,33.070,156.081
C07947=1066.633,328.717,399.960,174.259,33.075,156.082
C07948=1066.640,328.965,399.926,174.262,33.080,156.083
C07949=1066.646,329.212,399.892,174.266,33.085,156.084
C07950=1066.652,329.460,399.858,174.269,33.089,156.085
C07951=1066.659,329.707,399.824,174.272,33.094,156.086
C07952=1066.665,329.955,399.790,174.276,33.099,156.087
C07953=1066.672,330.202,399.755,174.279,33.103,156.088
C07954=1066.679,330.449,399.721,174.283,33.108,156.089
C07955=1066.685,330.697,399.687,174.286,33.113,156.089
C07956=1066.691,330.929,399.656,174.289,33.117,156.090
C07957=1066.697,331.160,399.623,174.292,33.122,156.091
C07958=1066.703,331.391,399.591,174.296,33.126,156.092
C07959=1066.708,331.621,399.559,174.299,33.131,156.093
C07960=1066.715,331.853,399.527,174.302,33.136,156.094
C07961=1066.721,332.084,399.495,174.305,33.140,156.095
C07962=1066.726,332.315,399.462,174.308,33.144,156.096
C07963=1066.732,332.547,399.430,174.312,33.149,156.097
C07964=1066.738,332.794,399.396,174.315,33.154,156.098
C07965=1066.745,333.041,399.361,174.318,33.159,156.099
C07966=1066.751,333.289,399.326,174.323,33.164,156.100
C07967=1066.757,333.536,399.292,174.326,33.169,156.101
C07968=1066.764,333.784,399.257,174.330,33.173,156.102
C07969=1066.771,334.032,399.223,174.333,33.178,156.102
C07970=1066.776,334.279,399.189,174.337,33.184,156.104
C07971=1066.783,334.526,399.153,174.340,33.188,156.104
C07972=1066.790,334.774,399.119,174.344,33.193,156.105
C07973=1066.796,335.022,399.084,174.347,33.198,156.106
C07974=1066.802,335.269,399.050,174.351,33.203,156.107
C07975=1066.809,335.516,399.015,174.354,33.208,156.108
C07976=1066.816,335.764,398.980,174.358,33.213,156.109
C07977=1066.822,336.012,398.945,174.361,33.218,156.110
C07978=1066.828,336.259,398.911,174.365,33.223,156.111
C07979=1066.835,336.506,398.876,174.368,33.228,156.112
C07980=1066.842,336.754,398.841,174.371,33.232,156.113
C07981=1066.848,337.002,398.806,174.375,33.238,156.114
C07982=1066.855,337.249,398.771,174.379,33.243,156.115
C07983=1066.860,337.497,398.737,174.382,33.248,156.116
C07984=1066.867,337.744,398.701,174.385,33.253,156.117
C07985=1066.874,337.991,398.666,174.390,33.258,156.118
C07986=1066.880,338.239,398.632,174.394,33.263,156.119
C07987=1066.886,338.487,398.596,174.397,33.268,156.121
C07988=1066.892,338.734,398.561,174.401,33.273,156.121
C07989=1066.899,338.981,398.526,174.404,33.278,156.123
C07990=1066.906,339.229,398.491,174.408,33.283,156.124
C07991=1066.911,339.477,398.456,174.411,33.288,156.125
C07992=1066.918,339.724,398.421,174.415,33.293,156.126
C07993=1066.925,339.972,398.386,174.418,33.298,156.127
C07994=1066.930,340.219,398.351,174.422,33.303,156.128
C07995=1066.937,340.466,398.315,174.425,33.308,156.129
C07996=1066.944,340.713,398.280,174.429,33.313,156.130
C07997=1066.950,340.961,398.245,174.432,33.318,156.131
C07998=1066.957,341.208,398.209,174.436,33.324,156.132
C07999=1066.964,341.456,398.174,174.440,33.329,156.133
C08000=1066.969,341.704,398.139,174.444,33.334,156.134
C08001=1066.976,341.951,398.104,174.448,33.339,156.135
C08002=1066.983,342.199,398.069,174.451,33.344,156.136
C08003=1066.989,342.446,398.033,174.455,33.349,156.137
C08004=1066.996,342.693,397.997,174.458,33.354,156.138
C08005=1067.003,342.940,397.962,174.462,33.360,156.139
C08006=1067.009,343.188,397.927,174.465,33.365,156.140
C08007=1067.015,343.436,397.891,174.469,33.370,156.141
C08008=1067.022,343.683,397.856,174.473,33.375,156.142
C08009=1067.028,343.931,397.821,174.476,33.380,156.143
C08010=1067.035,344.178,397.785,174.481,33.385,156.144
C08011=1067.041,344.426,397.750,174.484,33.391,156.145
C08012=1067.047,344.654,397.717,174.488,33.395,156.146
C08013=1067.052,344.882,397.684,174.491,33.401,156.147
C08014=1067.059,345.111,397.651,174.494,33.405,156.148
C08015=1067.065,345.339,397.618,174.498,33.410,156.149
C08016=1067.071,345.569,397.585,174.501,33.415,156.150
C08017=1067.077,345.797,397.552,174.504,33.420,156.151
C08018=1067.083,346.026,397.518,174.508,33.425,156.152
C08019=1067.089,346.254,397.486,174.511,33.430,156.153
C08020=1067.095,346.502,397.450,174.515,33.435,156.155
C08021=1067.102,346.749,397.414,174.519,33.440,156.156
C08022=1067.108,346.996,397.378,174.523,33.446,156.157
C08023=1067.114,347.243,397.342,174.527,33.451,156.158
C08024=1067.121,347.491,397.307,174.530,33.456,156.159
C08025=1067.128,347.739,397.271,174.534,33.461,156.160
C08026=1067.135,347.986,397.235,174.538,33.467,156.161
C08027=1067.141,348.234,397.199,174.541,33.472,156.162
C08028=1067.147,348.481,397.163,174.545,33.478,156.163
C08029=1067.154,348.728,397.126,174.549,33.483,156.164
C08030=1067.160,348.975,397.091,174.553,33.488,156.165
C08031=1067.167,349.222,397.055,174.557,33.494,156.167
C08032=1067.173,349.470,397.019,174.561,33.499,156.168
C08033=1067.180,349.717,396.983,174.564,33.504,156.169
C08034=1067.187,349.964,396.946,174.568,33.510,156.170
C08035=1067.193,350.212,396.911,174.572,33.516,156.171
C08036=1067.200,350.459,396.875,174.575,33.521,156.172
C08037=1067.206,350.706,396.838,174.579,33.526,156.173
C08038=1067.213,350.954,396.802,174.584,33.532,156.174
C08039=1067.219,351.201,396.766,174.588,33.537,156.176
C08040=1067.226,351.448,396.730,174.591,33.542,156.177
C08041=1067.233,351.695,396.693,174.595,33.548,156.178
C08042=1067.239,351.943,396.657,174.599,33.553,156.179
C08043=1067.245,352.190,396.621,174.602,33.559,156.180
C08044=1067.252,352.438,396.585,174.606,33.564,156.181
C08045=1067.259,352.684,396.549,174.611,33.570,156.182
C08046=1067.265,352.931,396.512,174.615,33.575,156.183
C08047=1067.272,353.179,396.475,174.618,33.581,156.185
C08048=1067.279,353.426,396.439,174.622,33.586,156.186
C08049=1067.285,353.673,396.403,174.626,33.592,156.187
C08050=1067.292,353.921,396.366,174.630,33.598,156.188
C08051=1067.298,354.168,396.329,174.633,33.603,156.189
C08052=1067.304,354.415,396.293,174.638,33.609,156.190
C08053=1067.311,354.662,396.256,174.642,33.615,156.192
C08054=1067.318,354.910,396.220,174.646,33.620,156.193
C08055=1067.324,355.157,396.183,174.649,33.626,156.194
C08056=1067.330,355.404,396.147,174.653,33.632,156.195
C08057=1067.337,355.652,396.110,174.657,33.637,156.196
C08058=1067.344,355.899,396.073,174.661,33.643,156.197
C08059=1067.350,356.146,396.037,174.665,33.648,156.199
C08060=1067.357,356.393,395.999,174.669,33.654,156.200
C08061=1067.364,356.640,395.963,174.673,33.660,156.201
C08062=1067.371,356.888,395.926,174.677,33.666,156.202
C08063=1067.377,357.135,395.890,174.681,33.671,156.203
C08064=1067.384,357.381,395.853,174.684,33.677,156.205
C08065=1067.390,357.629,395.816,174.689,33.682,156.206
C08066=1067.397,357.876,395.779,174.693,33.688,156.207
C08067=1067.404,358.123,395.742,174.697,33.694,156.208
C08068=1067.414,358.502,395.686,174.703,33.703,156.210
C08069=1067.425,358.881,395.629,174.710,33.711,156.212
C08070=1067.434,359.260,395.573,174.716,33.721,156.214
C08071=1067.445,359.638,395.515,174.721,33.729,156.216
C08072=1067.451,359.885,395.479,174.725,33.735,156.217
C08073=1067.458,360.133,395.441,174.729,33.741,156.218
C08074=1067.465,360.380,395.405,174.734,33.747,156.219
C08075=1067.471,360.627,395.367,174.738,33.753,156.221
C08076=1067.478,360.874,395.330,174.742,33.759,156.222
C08077=1067.485,361.121,395.293,174.746,33.764,156.223
C08078=1067.491,361.368,395.256,174.749,33.770,156.224
C08079=1067.498,361.616,395.218,174.754,33.776,156.226
C08080=1067.504,361.862,395.181,174.758,33.782,156.227
C08081=1067.511,362.110,395.144,174.762,33.788,156.228
C08082=1067.518,362.356,395.107,174.766,33.794,156.229
C08083=1067.524,362.604,395.069,174.770,33.800,156.231
C08084=1067.532,362.851,395.031,174.775,33.806,156.232
C08085=1067.538,363.098,394.995,174.779,33.811,156.233
C08086=1067.545,363.345,394.957,174.783,33.818,156.234
C08087=1067.551,363.592,394.920,174.786,33.823,156.236
C08088=1067.558,363.839,394.882,174.791,33.830,156.237
C08089=1067.566,364.086,394.844,174.795,33.835,156.238
C08090=1067.572,364.333,394.807,174.799,33.842,156.239
C08091=1067.579,364.581,394.770,174.803,33.847,156.241
C08092=1067.588,364.910,394.720,174.808,33.855,156.242
C08093=1067.596,365.239,394.669,174.815,33.864,156.244
C08094=1067.605,365.569,394.619,174.820,33.872,156.246
C08095=1067.614,365.899,394.568,174.825,33.880,156.248
C08096=1067.621,366.146,394.531,174.830,33.886,156.249
C08097=1067.627,366.392,394.493,174.834,33.893,156.250
C08098=1067.634,366.639,394.455,174.838,33.898,156.252
C08099=1067.641,366.886,394.417,174.842,33.905,156.253
C08100=1067.648,367.133,394.380,174.847,33.911,156.254
C08101=1067.654,367.380,394.341,174.851,33.917,156.256
C08102=1067.661,367.627,394.304,174.855,33.923,156.257
C08103=1067.668,367.875,394.266,174.859,33.929,156.258
C08104=1067.674,368.121,394.227,174.864,33.935,156.260
C08105=1067.681,368.368,394.190,174.868,33.942,156.261
C08106=1067.688,368.616,394.152,174.872,33.948,156.262
C08107=1067.695,368.862,394.113,174.876,33.954,156.264
C08108=1067.701,369.109,394.076,174.881,33.961,156.265
C08109=1067.708,369.356,394.038,174.885,33.967,156.266
C08110=1067.715,369.603,393.999,174.889,33.973,156.268
C08111=1067.722,369.850,393.961,174.893,33.979,156.269
C08112=1067.729,370.097,393.924,174.898,33.986,156.270
C08113=1067.736,370.344,393.885,174.902,33.992,156.272
C08114=1067.742,370.591,393.848,174.906,33.998,156.273
C08115=1067.749,370.837,393.809,174.911,34.004,156.274
C08116=1067.756,371.085,393.771,174.915,34.011,156.276
C08117=1067.763,371.331,393.732,174.919,34.017,156.277
C08118=1067.770,371.579,393.694,174.923,34.024,156.279
C08119=1067.777,371.826,393.656,174.928,34.030,156.280
C08120=1067.784,372.065,393.619,174.932,34.036,156.281
C08121=1067.790,372.304,393.581,174.936,34.042,156.283
C08122=1067.797,372.544,393.544,174.940,34.049,156.284
C08123=1067.804,372.783,393.507,174.945,34.055,156.285
C08124=1067.811,373.022,393.470,174.949,34.061,156.287
C08125=1067.817,373.261,393.433,174.953,34.067,156.288
C08126=1067.823,373.500,393.395,174.958,34.074,156.289
C08127=1067.830,373.740,393.358,174.962,34.080,156.291
C08128=1067.836,373.986,393.319,174.966,34.087,156.292
C08129=1067.843,374.233,393.281,174.971,34.093,156.294
C08130=1067.850,374.480,393.242,174.975,34.100,156.295
C08131=1067.857,374.727,393.203,174.979,34.106,156.297
C08132=1067.864,374.974,393.164,174.983,34.113,156.298
C08133=1067.871,375.220,393.126,174.988,34.119,156.299
C08134=1067.878,375.467,393.087,174.992,34.126,156.301
C08135=1067.885,375.714,393.048,174.996,34.133,156.302
C08136=1067.892,375.961,393.009,175.002,34.139,156.304
C08137=1067.899,376.208,392.970,175.006,34.146,156.305
C08138=1067.905,376.454,392.932,175.010,34.153,156.307
C08139=1067.912,376.701,392.893,175.015,34.160,156.308
C08140=1067.919,376.948,392.854,175.019,34.166,156.310
C08141=1067.926,377.195,392.815,175.023,34.173,156.311
C08142=1067.933,377.442,392.776,175.028,34.179,156.312
C08143=1067.939,377.688,392.737,175.033,34.186,156.314
C08144=1067.947,377.936,392.698,175.037,34.193,156.315
C08145=1067.954,378.182,392.659,175.042,34.200,156.317
C08146=1067.961,378.429,392.620,175.046,34.206,156.318
C08147=1067.968,378.676,392.581,175.051,34.213,156.320
C08148=1067.974,378.923,392.542,175.055,34.220,156.321
C08149=1067.981,379.169,392.503,175.060,34.227,156.323
C08150=1067.988,379.416,392.464,175.065,34.234,156.324
C08151=1067.996,379.663,392.425,175.069,34.241,156.326
C08152=1068.003,379.909,392.385,175.073,34.247,156.327
C08153=1068.010,380.156,392.346,175.079,34.254,156.329
C08154=1068.017,380.402,392.307,175.083,34.261,156.330
C08155=1068.024,380.650,392.267,175.087,34.268,156.332
C08156=1068.031,380.897,392.229,175.092,34.275,156.334
C08157=1068.038,381.143,392.189,175.096,34.282,156.335
C08158=1068.045,381.390,392.150,175.102,34.289,156.337
C08159=1068.052,381.637,392.110,175.106,34.296,156.338
C08160=1068.059,381.883,392.070,175.110,34.303,156.340
C08161=1068.066,382.130,392.031,175.115,34.310,156.341
C08162=1068.072,382.377,391.991,175.120,34.317,156.343
C08163=1068.080,382.624,391.952,175.125,34.324,156.344
C08164=1068.087,382.870,391.912,175.129,34.331,156.346
C08165=1068.093,383.117,391.872,175.133,34.338,156.348
C08166=1068.100,383.363,391.833,175.139,34.345,156.349
C08167=1068.108,383.611,391.793,175.143,34.352,156.351
C08168=1068.114,383.857,391.753,175.148,34.360,156.352
C08169=1068.121,384.103,391.714,175.153,34.367,156.354
C08170=1068.129,384.350,391.674,175.158,34.374,156.356
C08171=1068.135,384.597,391.634,175.162,34.381,156.357
C08172=1068.142,384.843,391.594,175.166,34.388,156.359
C08173=1068.149,385.090,391.554,175.172,34.395,156.360
C08174=1068.156,385.336,391.514,175.176,34.403,156.362
C08175=1068.164,385.584,391.475,175.181,34.410,156.364
C08176=1068.171,385.845,391.432,175.186,34.418,156.365
C08177=1068.178,386.107,391.390,175.192,34.425,156.367
C08178=1068.187,386.369,391.347,175.196,34.433,156.369
C08179=1068.193,386.631,391.305,175.202,34.441,156.371
C08180=1068.201,386.877,391.265,175.206,34.448,156.372
C08181=1068.208,387.124,391.225,175.211,34.456,156.374
C08182=1068.215,387.371,391.185,175.216,34.463,156.375
C08183=1068.222,387.616,391.144,175.220,34.470,156.377
C08184=1068.229,387.864,391.104,175.226,34.478,156.379
C08185=1068.237,388.110,391.064,175.230,34.485,156.380
C08186=1068.244,388.357,391.024,175.236,34.492,156.382
C08187=1068.251,388.603,390.984,175.240,34.500,156.384
C08188=1068.259,388.850,390.944,175.245,34.507,156.385
C08189=1068.265,389.096,390.904,175.250,34.515,156.387
C08190=1068.273,389.342,390.863,175.255,34.522,156.389
C08191=1068.280,389.590,390.822,175.260,34.530,156.390
C08192=1068.287,389.836,390.783,175.265,34.537,156.392
C08193=1068.295,390.082,390.742,175.270,34.545,156.394
C08194=1068.302,390.329,390.702,175.275,34.552,156.396
C08195=1068.309,390.575,390.661,175.280,34.560,156.397
C08196=1068.317,390.822,390.621,175.285,34.567,156.399
C08197=1068.323,391.068,390.580,175.289,34.575,156.401
C08198=1068.330,391.315,390.540,175.295,34.583,156.402
C08199=1068.338,391.561,390.499,175.299,34.591,156.404
C08200=1068.345,391.807,390.458,175.305,34.598,156.406
C08201=1068.352,392.055,390.418,175.309,34.605,156.408
C08202=1068.360,392.301,390.377,175.315,34.613,156.409
C08203=1068.367,392.547,390.336,175.319,34.621,156.411
C08204=1068.374,392.794,390.296,175.325,34.629,156.413
C08205=1068.381,393.041,390.254,175.330,34.637,156.415
C08206=1068.388,393.286,390.214,175.335,34.645,156.417
C08207=1068.396,393.533,390.173,175.340,34.652,156.418
C08208=1068.403,393.779,390.132,175.345,34.660,156.420
C08209=1068.410,394.027,390.091,175.350,34.668,156.422
C08210=1068.417,394.273,390.050,175.355,34.676,156.424
C08211=1068.425,394.519,390.010,175.360,34.684,156.426
C08212=1068.432,394.765,389.968,175.365,34.692,156.427
C08213=1068.439,395.012,389.927,175.371,34.700,156.429
C08214=1068.447,395.259,389.886,175.376,34.708,156.431
C08215=1068.454,395.505,389.845,175.381,34.716,156.433
C08216=1068.461,395.751,389.804,175.386,34.724,156.435
C08217=1068.468,395.998,389.763,175.391,34.732,156.437
C08218=1068.475,396.244,389.721,175.396,34.740,156.438
C08219=1068.483,396.490,389.679,175.402,34.748,156.440
C08220=1068.490,396.737,389.638,175.407,34.756,156.442
C08221=1068.497,396.983,389.597,175.412,34.764,156.444
C08222=1068.505,397.230,389.556,175.417,34.772,156.446
C08223=1068.513,397.476,389.515,175.422,34.780,156.448
C08224=1068.520,397.722,389.473,175.428,34.789,156.450
C08225=1068.527,397.969,389.432,175.433,34.797,156.451
C08226=1068.535,398.215,389.391,175.438,34.805,156.453
C08227=1068.542,398.462,389.348,175.444,34.813,156.455
C08228=1068.549,398.708,389.307,175.449,34.822,156.457
C08229=1068.556,398.954,389.265,175.454,34.830,156.459
C08230=1068.564,399.201,389.224,175.460,34.838,156.461
C08231=1068.571,399.447,389.182,175.464,34.846,156.463
C08232=1068.579,399.725,389.135,175.471,34.856,156.465
C08233=1068.588,400.003,389.088,175.477,34.865,156.467
C08234=1068.596,400.281,389.041,175.483,34.875,156.469
C08235=1068.605,400.558,388.994,175.489,34.884,156.472
C08236=1068.612,400.804,388.952,175.494,34.893,156.474
C08237=1068.619,401.051,388.910,175.500,34.901,156.476
C08238=1068.626,401.297,388.868,175.505,34.910,156.478
C08239=1068.635,401.544,388.826,175.510,34.918,156.480
C08240=1068.642,401.790,388.784,175.516,34.927,156.482
C08241=1068.650,402.037,388.743,175.522,34.935,156.483
C08242=1068.656,402.283,388.700,175.527,34.944,156.485
C08243=1068.664,402.529,388.658,175.532,34.952,156.488
C08244=1068.672,402.775,388.616,175.538,34.961,156.489
C08245=1068.680,403.021,388.574,175.543,34.969,156.491
C08246=1068.687,403.268,388.532,175.549,34.978,156.494
C08247=1068.694,403.514,388.490,175.554,34.987,156.496
C08248=1068.702,403.761,388.448,175.560,34.995,156.498
C08249=1068.709,404.007,388.406,175.565,35.004,156.500
C08250=1068.717,404.253,388.364,175.571,35.013,156.502
C08251=1068.725,404.499,388.321,175.577,35.022,156.504
C08252=1068.732,404.746,388.278,175.582,35.031,156.506
C08253=1068.739,404.992,388.236,175.587,35.039,156.508
C08254=1068.747,405.239,388.193,175.593,35.048,156.510
C08255=1068.755,405.485,388.151,175.599,35.057,156.512
C08256=1068.761,405.731,388.109,175.605,35.066,156.514
C08257=1068.770,405.977,388.066,175.611,35.075,156.516
C08258=1068.777,406.223,388.023,175.616,35.084,156.518
C08259=1068.785,406.470,387.981,175.621,35.093,156.521
C08260=1068.792,406.716,387.938,175.627,35.102,156.523
C08261=1068.800,406.962,387.895,175.633,35.111,156.525
C08262=1068.807,407.208,387.853,175.639,35.120,156.527
C08263=1068.814,407.454,387.809,175.645,35.129,156.529
C08264=1068.823,407.701,387.767,175.650,35.138,156.531
C08265=1068.830,407.946,387.724,175.656,35.148,156.533
C08266=1068.837,408.193,387.681,175.662,35.157,156.536
C08267=1068.845,408.439,387.638,175.668,35.166,156.538
C08268=1068.853,408.686,387.595,175.674,35.175,156.540
C08269=1068.860,408.931,387.552,175.680,35.184,156.542
C08270=1068.868,409.178,387.509,175.686,35.194,156.544
C08271=1068.876,409.425,387.466,175.691,35.203,156.547
C08272=1068.883,409.670,387.423,175.697,35.212,156.549
C08273=1068.891,409.916,387.380,175.703,35.222,156.551
C08274=1068.898,410.162,387.337,175.709,35.231,156.553
C08275=1068.906,410.409,387.294,175.715,35.240,156.555
C08276=1068.914,410.655,387.251,175.721,35.250,156.558
C08277=1068.922,410.901,387.207,175.727,35.259,156.560
C08278=1068.929,411.147,387.164,175.733,35.269,156.562
C08279=1068.937,411.393,387.120,175.739,35.278,156.564
C08280=1068.945,411.639,387.078,175.745,35.288,156.567
C08281=1068.953,411.885,387.034,175.751,35.297,156.569
C08282=1068.961,412.131,386.990,175.757,35.306,156.571
C08283=1068.968,412.378,386.947,175.763,35.316,156.574
C08284=1068.976,412.623,386.904,175.769,35.326,156.576
C08285=1068.984,412.869,386.860,175.776,35.335,156.578
C08286=1068.992,413.116,386.817,175.781,35.345,156.581
C08287=1068.999,413.362,386.773,175.787,35.355,156.583
C08288=1069.008,413.644,386.723,175.795,35.366,156.586
C08289=1069.018,413.926,386.673,175.802,35.377,156.588
C08290=1069.027,414.208,386.623,175.809,35.388,156.591
C08291=1069.036,414.489,386.573,175.816,35.399,156.594
C08292=1069.044,414.735,386.530,175.822,35.409,156.596
C08293=1069.052,414.981,386.486,175.828,35.419,156.598
C08294=1069.060,415.227,386.442,175.834,35.429,156.601
C08295=1069.067,415.473,386.397,175.840,35.439,156.603
C08296=1069.075,415.720,386.354,175.847,35.449,156.606
C08297=1069.083,415.965,386.309,175.853,35.459,156.608
C08298=1069.091,416.211,386.265,175.859,35.469,156.611
C08299=1069.099,416.458,386.221,175.866,35.479,156.613
C08300=1069.107,416.703,386.177,175.873,35.489,156.615
C08301=1069.115,416.949,386.133,175.879,35.499,156.618
C08302=1069.123,417.195,386.089,175.885,35.509,156.620
C08303=1069.131,417.441,386.045,175.892,35.519,156.623
C08304=1069.139,417.687,386.000,175.898,35.530,156.625
C08305=1069.147,417.933,385.956,175.904,35.540,156.628
C08306=1069.154,418.179,385.911,175.911,35.550,156.630
C08307=1069.162,418.424,385.867,175.917,35.561,156.633
C08308=1069.170,418.671,385.823,175.924,35.571,156.635
C08309=1069.178,418.917,385.779,175.931,35.581,156.638
C08310=1069.186,419.162,385.735,175.937,35.592,156.640
C08311=1069.194,419.408,385.690,175.943,35.602,156.643
C08312=1069.203,419.654,385.645,175.950,35.612,156.645
C08313=1069.211,419.900,385.600,175.956,35.623,156.648
C08314=1069.219,420.146,385.556,175.964,35.634,156.651
C08315=1069.227,420.391,385.511,175.970,35.644,156.653
C08316=1069.235,420.637,385.467,175.977,35.654,156.656
C08317=1069.244,420.884,385.422,175.983,35.665,156.658
C08318=1069.251,421.129,385.377,175.991,35.676,156.661
C08319=1069.259,421.375,385.332,175.997,35.686,156.664
C08320=1069.268,421.621,385.288,176.004,35.697,156.666
C08321=1069.276,421.867,385.242,176.010,35.708,156.669
C08322=1069.284,422.112,385.198,176.018,35.719,156.672
C08323=1069.291,422.358,385.152,176.024,35.729,156.674
C08324=1069.300,422.604,385.107,176.031,35.740,156.677
C08325=1069.308,422.850,385.062,176.037,35.751,156.680
C08326=1069.316,423.095,385.017,176.045,35.762,156.682
C08327=1069.325,423.341,384.972,176.051,35.773,156.685
C08328=1069.332,423.587,384.926,176.058,35.784,156.688
C08329=1069.340,423.832,384.882,176.066,35.795,156.690
C08330=1069.349,424.079,384.836,176.072,35.806,156.693
C08331=1069.357,424.324,384.791,176.079,35.817,156.696
C08332=1069.365,424.570,384.745,176.086,35.828,156.699
C08333=1069.374,424.815,384.700,176.093,35.840,156.702
C08334=1069.382,425.062,384.654,176.101,35.851,156.704
C08335=1069.390,425.307,384.609,176.107,35.862,156.707
C08336=1069.398,425.553,384.563,176.114,35.873,156.710
C08337=1069.407,425.798,384.518,176.122,35.884,156.713
C08338=1069.415,426.044,384.472,176.129,35.896,156.715
C08339=1069.423,426.289,384.427,176.136,35.907,156.718
C08340=1069.431,426.536,384.381,176.143,35.918,156.721
C08341=1069.441,426.781,384.335,176.151,35.929,156.724
C08342=1069.448,427.026,384.289,176.158,35.941,156.727
C08343=1069.457,427.272,384.244,176.165,35.952,156.730
C08344=1069.468,427.573,384.187,176.173,35.966,156.733
C08345=1069.478,427.874,384.131,176.182,35.980,156.737
C08346=1069.488,428.175,384.075,176.192,35.995,156.740
C08347=1069.498,428.475,384.018,176.201,36.009,156.744
C08348=1069.506,428.721,383.972,176.208,36.021,156.747
C08349=1069.515,428.966,383.926,176.215,36.032,156.750
C08350=1069.523,429.213,383.880,176.223,36.044,156.753
C08351=1069.532,429.458,383.834,176.230,36.056,156.756
C08352=1069.540,429.703,383.788,176.238,36.068,156.759
C08353=1069.548,429.949,383.741,176.245,36.080,156.762
C08354=1069.557,430.194,383.694,176.253,36.092,156.765
C08355=1069.565,430.440,383.648,176.261,36.103,156.768
C08356=1069.574,430.686,383.602,176.268,36.115,156.771
C08357=1069.583,430.931,383.556,176.276,36.127,156.774
C08358=1069.591,431.176,383.509,176.283,36.139,156.777
C08359=1069.599,431.421,383.463,176.291,36.151,156.780
C08360=1069.608,431.667,383.416,176.299,36.163,156.783
C08361=1069.616,431.912,383.369,176.307,36.176,156.786
C08362=1069.625,432.158,383.322,176.314,36.188,156.789
C08363=1069.634,432.403,383.276,176.322,36.201,156.792
C08364=1069.642,432.649,383.229,176.330,36.213,156.796
C08365=1069.651,432.894,383.182,176.337,36.225,156.799
C08366=1069.659,433.139,383.135,176.345,36.238,156.802
C08367=1069.668,433.385,383.088,176.353,36.250,156.805
C08368=1069.677,433.630,383.041,176.361,36.262,156.808
C08369=1069.685,433.875,382.994,176.369,36.275,156.811
C08370=1069.694,434.121,382.947,176.376,36.287,156.815
C08371=1069.703,434.366,382.900,176.385,36.300,156.818
C08372=1069.711,434.612,382.852,176.393,36.313,156.821
C08373=1069.719,434.857,382.806,176.401,36.325,156.824
C08374=1069.728,435.102,382.758,176.409,36.338,156.828
C08375=1069.737,435.347,382.711,176.417,36.351,156.831
C08376=1069.746,435.593,382.664,176.425,36.363,156.834
C08377=1069.755,435.838,382.616,176.433,36.376,156.838
C08378=1069.764,436.083,382.569,176.441,36.389,156.841
C08379=1069.772,436.328,382.522,176.449,36.402,156.844
C08380=1069.781,436.574,382.474,176.458,36.415,156.848
C08381=1069.790,436.819,382.426,176.466,36.428,156.851
C08382=1069.799,437.064,382.379,176.474,36.441,156.854
C08383=1069.808,437.309,382.331,176.483,36.454,156.858
C08384=1069.817,437.554,382.283,176.491,36.467,156.861
C08385=1069.826,437.799,382.236,176.499,36.480,156.864
C08386=1069.835,438.045,382.188,176.508,36.493,156.868
C08387=1069.843,438.290,382.140,176.516,36.506,156.871
C08388=1069.852,438.535,382.093,176.525,36.519,156.875
C08389=1069.862,438.781,382.045,176.533,36.533,156.878
C08390=1069.870,439.025,381.996,176.541,36.546,156.882
C08391=1069.880,439.271,381.948,176.550,36.559,156.885
C08392=1069.888,439.516,381.901,176.559,36.573,156.889
C08393=1069.897,439.761,381.852,176.568,36.587,156.892
C08394=1069.906,440.006,381.804,176.576,36.600,156.896
C08395=1069.915,440.251,381.755,176.585,36.613,156.899
C08396=1069.924,440.496,381.708,176.593,36.627,156.903
C08397=1069.934,440.741,381.659,176.602,36.641,156.907
C08398=1069.942,440.986,381.611,176.611,36.655,156.910
C08399=1069.952,441.231,381.563,176.620,36.668,156.914
C08400=1069.959,441.446,381.520,176.628,36.680,156.917
C08401=1069.967,441.661,381.478,176.636,36.693,156.920
C08402=1069.975,441.875,381.435,176.643,36.705,156.923
C08403=1069.984,442.090,381.392,176.651,36.717,156.927
C08404=1069.992,442.305,381.350,176.659,36.729,156.930
C08405=1069.999,442.520,381.307,176.667,36.741,156.933
C08406=1070.007,442.734,381.264,176.675,36.754,156.936
C08407=1070.016,442.949,381.221,176.683,36.766,156.940
C08408=1070.024,443.193,381.173,176.691,36.780,156.943
C08409=1070.034,443.438,381.124,176.701,36.794,156.947
C08410=1070.043,443.684,381.075,176.710,36.808,156.951
C08411=1070.052,443.929,381.026,176.720,36.823,156.955
C08412=1070.062,444.173,380.977,176.728,36.837,156.959
C08413=1070.071,444.418,380.928,176.738,36.851,156.962
C08414=1070.080,444.663,380.879,176.747,36.866,156.966
C08415=1070.090,444.908,380.830,176.757,36.881,156.970
C08416=1070.099,445.153,380.780,176.766,36.895,156.974
C08417=1070.108,445.397,380.731,176.776,36.910,156.978
C08418=1070.117,445.643,380.681,176.784,36.924,156.982
C08419=1070.127,445.887,380.632,176.794,36.939,156.986
C08420=1070.136,446.132,380.582,176.803,36.954,156.990
C08421=1070.145,446.377,380.533,176.813,36.968,156.994
C08422=1070.155,446.622,380.483,176.823,36.983,156.998
C08423=1070.164,446.866,380.434,176.832,36.998,157.002
C08424=1070.174,447.111,380.384,176.842,37.013,157.006
C08425=1070.183,447.355,380.335,176.852,37.028,157.010
C08426=1070.192,447.601,380.285,176.861,37.043,157.014
C08427=1070.202,447.846,380.235,176.871,37.058,157.018
C08428=1070.212,448.089,380.186,176.881,37.073,157.022
C08429=1070.222,448.332,380.136,176.891,37.088,157.026
C08430=1070.233,448.577,380.087,176.899,37.102,157.030
C08431=1070.245,448.822,380.039,176.908,37.117,157.034
C08432=1070.259,449.066,379.992,176.916,37.130,157.037
C08433=1070.273,449.311,379.945,176.925,37.143,157.041
C08434=1070.289,449.556,379.899,176.933,37.156,157.044
C08435=1070.306,449.802,379.854,176.940,37.168,157.048
C08436=1069.957,449.802,379.601,176.927,37.307,157.085
C08437=1069.941,449.557,379.646,176.920,37.295,157.081
C08438=1069.925,449.312,379.692,176.911,37.282,157.078
C08439=1069.911,449.067,379.739,176.903,37.269,157.074
C08440=1069.897,448.822,379.786,176.894,37.255,157.071
C08441=1069.885,448.577,379.835,176.886,37.241,157.067
C08442=1069.873,448.332,379.884,176.876,37.227,157.063
C08443=1069.863,448.088,379.932,176.866,37.212,157.059
C08444=1069.853,447.845,379.982,176.856,37.197,157.055
C08445=1069.843,447.601,380.032,176.847,37.182,157.051
C08446=1069.834,447.356,380.082,176.837,37.167,157.047
C08447=1069.825,447.111,380.131,176.827,37.152,157.043
C08448=1069.815,446.867,380.181,176.817,37.137,157.039
C08449=1069.806,446.622,380.231,176.807,37.122,157.035
C08450=1069.795,446.377,380.281,176.798,37.108,157.031
C08451=1069.786,446.132,380.330,176.788,37.093,157.027
C08452=1069.777,445.887,380.380,176.778,37.078,157.023
C08453=1069.768,445.642,380.429,176.769,37.063,157.019
C08454=1069.758,445.398,380.479,176.759,37.049,157.015
C08455=1069.749,445.153,380.528,176.749,37.034,157.011
C08456=1069.739,444.908,380.578,176.741,37.020,157.007
C08457=1069.730,444.663,380.627,176.731,37.005,157.003
C08458=1069.721,444.419,380.676,176.722,36.991,156.999
C08459=1069.712,444.174,380.725,176.712,36.977,156.995
C08460=1069.703,443.929,380.775,176.703,36.962,156.991
C08461=1069.693,443.684,380.823,176.693,36.948,156.988
C08462=1069.684,443.439,380.872,176.685,36.934,156.984
C08463=1069.675,443.194,380.921,176.675,36.920,156.980
C08464=1069.665,442.949,380.970,176.666,36.905,156.976
C08465=1069.650,442.539,381.052,176.651,36.882,156.970
C08466=1069.634,442.127,381.133,176.636,36.859,156.964
C08467=1069.619,441.717,381.215,176.621,36.835,156.958
C08468=1069.603,441.307,381.296,176.606,36.812,156.952
C08469=1069.594,441.062,381.345,176.596,36.798,156.948
C08470=1069.585,440.817,381.393,176.587,36.785,156.944
C08471=1069.577,440.572,381.442,176.579,36.771,156.941
C08472=1069.567,440.327,381.490,176.569,36.758,156.937
C08473=1069.558,440.082,381.539,176.561,36.744,156.933
C08474=1069.549,439.836,381.587,176.552,36.730,156.930
C08475=1069.541,439.592,381.636,176.544,36.717,156.926
C08476=1069.531,439.346,381.683,176.535,36.704,156.923
C08477=1069.522,439.101,381.731,176.526,36.690,156.919
C08478=1069.513,438.856,381.780,176.517,36.677,156.916
C08479=1069.504,438.611,381.827,176.509,36.663,156.912
C08480=1069.496,438.366,381.875,176.500,36.650,156.909
C08481=1069.486,438.121,381.924,176.492,36.637,156.905
C08482=1069.478,437.876,381.971,176.484,36.624,156.902
C08483=1069.468,437.630,382.019,176.475,36.611,156.899
C08484=1069.459,437.386,382.067,176.467,36.598,156.895
C08485=1069.450,437.140,382.114,176.457,36.585,156.892
C08486=1069.441,436.895,382.162,176.449,36.572,156.888
C08487=1069.433,436.650,382.210,176.441,36.559,156.885
C08488=1069.423,436.404,382.258,176.433,36.546,156.882
C08489=1069.415,436.159,382.304,176.424,36.533,156.878
C08490=1069.406,435.914,382.352,176.416,36.520,156.875
C08491=1069.397,435.669,382.399,176.408,36.508,156.872
C08492=1069.388,435.423,382.447,176.399,36.495,156.868
C08493=1069.379,435.178,382.494,176.391,36.482,156.865
C08494=1069.370,434.933,382.541,176.384,36.469,156.862
C08495=1069.362,434.688,382.589,176.376,36.457,156.858
C08496=1069.354,434.442,382.636,176.368,36.444,156.855
C08497=1069.345,434.197,382.684,176.359,36.432,156.852
C08498=1069.336,433.951,382.731,176.351,36.419,156.849
C08499=1069.327,433.706,382.778,176.343,36.407,156.846
C08500=1069.318,433.461,382.825,176.335,36.394,156.842
C08501=1069.310,433.215,382.872,176.327,36.382,156.839
C08502=1069.301,432.970,382.919,176.319,36.369,156.836
C08503=1069.292,432.725,382.966,176.312,36.357,156.833
C08504=1069.284,432.479,383.012,176.304,36.345,156.830
C08505=1069.275,432.234,383.059,176.296,36.332,156.826
C08506=1069.267,431.988,383.106,176.288,36.320,156.823
C08507=1069.258,431.743,383.153,176.281,36.308,156.820
C08508=1069.250,431.499,383.200,176.273,36.296,156.817
C08509=1069.241,431.253,383.246,176.265,36.284,156.814
C08510=1069.233,431.007,383.292,176.257,36.272,156.811
C08511=1069.225,430.761,383.339,176.250,36.260,156.808
C08512=1069.216,430.516,383.386,176.242,36.248,156.805
C08513=1069.208,430.270,383.433,176.234,36.236,156.802
C08514=1069.198,430.025,383.479,176.227,36.224,156.799
C08515=1069.190,429.779,383.525,176.219,36.212,156.796
C08516=1069.181,429.534,383.572,176.211,36.200,156.793
C08517=1069.173,429.289,383.618,176.204,36.188,156.790
C08518=1069.165,429.043,383.663,176.196,36.177,156.787
C08519=1069.156,428.797,383.710,176.188,36.165,156.784
C08520=1069.147,428.552,383.757,176.182,36.154,156.781
C08521=1069.138,428.250,383.814,176.172,36.139,156.777
C08522=1069.126,427.947,383.870,176.163,36.125,156.774
C08523=1069.117,427.644,383.926,176.154,36.111,156.770
C08524=1069.107,427.341,383.983,176.145,36.096,156.767
C08525=1069.098,427.096,384.029,176.137,36.085,156.764
C08526=1069.089,426.850,384.076,176.130,36.074,156.761
C08527=1069.081,426.605,384.121,176.123,36.062,156.758
C08528=1069.073,426.359,384.167,176.116,36.051,156.755
C08529=1069.064,426.113,384.212,176.108,36.040,156.752
C08530=1069.056,425.868,384.258,176.101,36.028,156.749
C08531=1069.047,425.622,384.303,176.094,36.017,156.747
C08532=1069.039,425.376,384.349,176.087,36.006,156.744
C08533=1069.030,425.130,384.394,176.079,35.995,156.741
C08534=1069.023,424.885,384.440,176.073,35.984,156.738
C08535=1069.014,424.639,384.485,176.066,35.973,156.735
C08536=1069.006,424.394,384.531,176.058,35.961,156.733
C08537=1068.997,424.148,384.576,176.052,35.950,156.730
C08538=1068.990,423.903,384.622,176.044,35.939,156.727
C08539=1068.981,423.656,384.667,176.037,35.928,156.724
C08540=1068.973,423.411,384.712,176.030,35.918,156.722
C08541=1068.964,423.165,384.758,176.023,35.906,156.719
C08542=1068.957,422.919,384.803,176.017,35.896,156.716
C08543=1068.949,422.674,384.848,176.009,35.885,156.714
C08544=1068.940,422.427,384.894,176.003,35.874,156.711
C08545=1068.932,422.182,384.938,175.996,35.863,156.708
C08546=1068.924,421.937,384.983,175.989,35.852,156.706
C08547=1068.916,421.690,385.028,175.982,35.842,156.703
C08548=1068.908,421.445,385.073,175.975,35.831,156.700
C08549=1068.900,421.199,385.118,175.968,35.820,156.698
C08550=1068.892,420.954,385.163,175.962,35.809,156.695
C08551=1068.883,420.707,385.208,175.955,35.799,156.692
C08552=1068.875,420.461,385.252,175.948,35.789,156.690
C08553=1068.868,420.215,385.297,175.941,35.778,156.687
C08554=1068.859,419.969,385.342,175.935,35.767,156.685
C08555=1068.851,419.724,385.387,175.928,35.757,156.682
C08556=1068.843,419.478,385.431,175.921,35.747,156.679
C08557=1068.835,419.232,385.476,175.914,35.736,156.677
C08558=1068.827,418.987,385.520,175.908,35.726,156.674
C08559=1068.819,418.740,385.565,175.902,35.716,156.672
C08560=1068.811,418.494,385.610,175.895,35.705,156.669
C08561=1068.803,418.248,385.654,175.888,35.695,156.667
C08562=1068.794,418.003,385.698,175.882,35.685,156.664
C08563=1068.786,417.757,385.743,175.875,35.675,156.662
C08564=1068.778,417.511,385.787,175.869,35.664,156.659
C08565=1068.771,417.265,385.831,175.863,35.654,156.657
C08566=1068.762,417.019,385.875,175.855,35.644,156.654
C08567=1068.755,416.773,385.920,175.849,35.634,156.652
C08568=1068.747,416.527,385.964,175.843,35.624,156.649
C08569=1068.739,416.281,386.008,175.836,35.614,156.647
C08570=1068.731,416.035,386.052,175.830,35.604,156.644
C08571=1068.723,415.789,386.097,175.824,35.593,156.642
C08572=1068.715,415.543,386.140,175.818,35.584,156.640
C08573=1068.707,415.297,386.185,175.811,35.574,156.637
C08574=1068.700,415.051,386.228,175.804,35.564,156.635
C08575=1068.692,414.805,386.273,175.798,35.554,156.632
C08576=1068.684,414.559,386.316,175.792,35.544,156.630
C08577=1068.675,414.276,386.366,175.785,35.533,156.627
C08578=1068.665,413.992,386.417,175.778,35.522,156.625
C08579=1068.656,413.708,386.467,175.771,35.510,156.622
C08580=1068.647,413.425,386.518,175.763,35.499,156.619
C08581=1068.639,413.179,386.561,175.757,35.489,156.617
C08582=1068.631,412.934,386.605,175.751,35.480,156.614
C08583=1068.623,412.687,386.649,175.745,35.470,156.612
C08584=1068.616,412.441,386.692,175.738,35.461,156.610
C08585=1068.607,412.195,386.735,175.732,35.451,156.608
C08586=1068.600,411.949,386.778,175.726,35.441,156.605
C08587=1068.592,411.703,386.822,175.720,35.432,156.603
C08588=1068.584,411.456,386.866,175.714,35.423,156.601
C08589=1068.576,411.210,386.909,175.708,35.413,156.598
C08590=1068.569,410.965,386.952,175.702,35.404,156.596
C08591=1068.561,410.718,386.996,175.696,35.394,156.594
C08592=1068.553,410.472,387.039,175.690,35.385,156.592
C08593=1068.545,410.227,387.082,175.684,35.375,156.589
C08594=1068.538,409.980,387.125,175.678,35.366,156.587
C08595=1068.530,409.733,387.168,175.672,35.357,156.585
C08596=1068.522,409.488,387.211,175.667,35.348,156.583
C08597=1068.515,409.242,387.255,175.661,35.338,156.580
C08598=1068.507,408.995,387.298,175.655,35.329,156.578
C08599=1068.499,408.749,387.340,175.649,35.320,156.576
C08600=1068.491,408.503,387.384,175.643,35.310,156.574
C08601=1068.485,408.257,387.426,175.637,35.301,156.572
C08602=1068.476,408.011,387.469,175.631,35.292,156.569
C08603=1068.469,407.765,387.513,175.625,35.283,156.567
C08604=1068.461,407.518,387.556,175.619,35.274,156.565
C08605=1068.454,407.273,387.598,175.613,35.265,156.563
C08606=1068.446,407.026,387.641,175.607,35.256,156.561
C08607=1068.438,406.780,387.684,175.602,35.246,156.559
C08608=1068.431,406.533,387.727,175.597,35.238,156.557
C08609=1068.424,406.287,387.769,175.591,35.229,156.554
C08610=1068.416,406.042,387.812,175.585,35.220,156.552
C08611=1068.408,405.795,387.855,175.579,35.211,156.550
C08612=1068.401,405.549,387.897,175.573,35.202,156.548
C08613=1068.393,405.302,387.940,175.567,35.193,156.546
C08614=1068.386,405.056,387.982,175.562,35.184,156.544
C08615=1068.378,404.810,388.024,175.557,35.175,156.542
C08616=1068.370,404.563,388.067,175.551,35.167,156.540
C08617=1068.363,404.317,388.109,175.545,35.158,156.538
C08618=1068.355,404.070,388.152,175.539,35.149,156.536
C08619=1068.348,403.824,388.194,175.533,35.140,156.533
C08620=1068.340,403.578,388.236,175.529,35.131,156.531
C08621=1068.333,403.332,388.278,175.523,35.123,156.529
C08622=1068.325,403.085,388.321,175.517,35.114,156.527
C08623=1068.318,402.839,388.363,175.511,35.106,156.525
C08624=1068.311,402.593,388.405,175.506,35.097,156.523
C08625=1068.303,402.346,388.448,175.501,35.088,156.521
C08626=1068.295,402.101,388.490,175.495,35.080,156.519
C08627=1068.288,401.854,388.531,175.489,35.071,156.517
C08628=1068.280,401.608,388.573,175.484,35.063,156.515
C08629=1068.273,401.362,388.615,175.479,35.054,156.513
C08630=1068.265,401.115,388.658,175.473,35.046,156.511
C08631=1068.258,400.868,388.699,175.467,35.037,156.509
C08632=1068.250,400.622,388.741,175.463,35.029,156.507
C08633=1068.242,400.343,388.788,175.456,35.019,156.505
C08634=1068.234,400.063,388.836,175.450,35.010,156.503
C08635=1068.225,399.784,388.884,175.444,35.000,156.501
C08636=1068.217,399.505,388.931,175.437,34.991,156.499
C08637=1068.209,399.258,388.972,175.433,34.983,156.497
C08638=1068.202,399.012,389.014,175.427,34.974,156.495
C08639=1068.194,398.766,389.055,175.421,34.966,156.493
C08640=1068.188,398.520,389.098,175.416,34.958,156.491
C08641=1068.180,398.273,389.139,175.411,34.949,156.489
C08642=1068.173,398.026,389.180,175.406,34.941,156.487
C08643=1068.165,397.780,389.222,175.400,34.933,156.485
C08644=1068.158,397.533,389.264,175.395,34.925,156.483
C08645=1068.150,397.287,389.305,175.390,34.917,156.481
C08646=1068.143,397.041,389.347,175.384,34.909,156.480
C08647=1068.136,396.795,389.388,175.380,34.900,156.478
C08648=1068.128,396.548,389.428,175.374,34.893,156.476
C08649=1068.121,396.302,389.469,175.368,34.884,156.474
C08650=1068.113,396.055,389.511,175.364,34.876,156.472
C08651=1068.106,395.809,389.553,175.358,34.869,156.470
C08652=1068.099,395.563,389.594,175.353,34.860,156.468
C08653=1068.091,395.316,389.635,175.348,34.853,156.467
C08654=1068.084,395.069,389.676,175.343,34.844,156.465
C08655=1068.077,394.823,389.718,175.338,34.837,156.463
C08656=1068.070,394.577,389.758,175.332,34.829,156.461
C08657=1068.063,394.330,389.800,175.327,34.821,156.459
C08658=1068.055,394.084,389.841,175.322,34.813,156.457
C08659=1068.047,393.837,389.881,175.317,34.805,156.456
C08660=1068.040,393.591,389.923,175.312,34.797,156.454
C08661=1068.034,393.344,389.963,175.307,34.789,156.452
C08662=1068.026,393.098,390.004,175.301,34.781,156.450
C08663=1068.018,392.851,390.045,175.297,34.774,156.448
C08664=1068.011,392.605,390.086,175.291,34.766,156.447
C08665=1068.004,392.359,390.127,175.287,34.758,156.445
C08666=1067.997,392.112,390.167,175.281,34.751,156.443
C08667=1067.989,391.865,390.208,175.276,34.743,156.441
C08668=1067.983,391.620,390.249,175.271,34.735,156.440
C08669=1067.976,391.372,390.289,175.266,34.727,156.438
C08670=1067.968,391.126,390.330,175.261,34.720,156.436
C08671=1067.961,390.880,390.371,175.256,34.712,156.434
C08672=1067.954,390.633,390.411,175.252,34.705,156.433
C08673=1067.946,390.387,390.452,175.246,34.697,156.431
C08674=1067.940,390.140,390.492,175.242,34.690,156.429
C08675=1067.932,389.894,390.533,175.236,34.682,156.428
C08676=1067.924,389.647,390.573,175.231,34.675,156.426
C08677=1067.917,389.401,390.614,175.226,34.667,156.424
C08678=1067.909,389.154,390.653,175.221,34.660,156.423
C08679=1067.902,388.907,390.694,175.217,34.652,156.421
C08680=1067.895,388.661,390.734,175.211,34.645,156.419
C08681=1067.888,388.414,390.775,175.207,34.637,156.417
C08682=1067.881,388.168,390.814,175.201,34.630,156.416
C08683=1067.874,387.921,390.856,175.197,34.622,156.414
C08684=1067.867,387.675,390.895,175.192,34.615,156.412
C08685=1067.860,387.428,390.936,175.187,34.608,156.411
C08686=1067.852,387.182,390.975,175.182,34.600,156.409
C08687=1067.845,386.935,391.015,175.177,34.593,156.407
C08688=1067.838,386.688,391.055,175.172,34.586,156.406
C08689=1067.830,386.425,391.098,175.167,34.578,156.404
C08690=1067.823,386.162,391.142,175.162,34.570,156.402
C08691=1067.816,385.898,391.184,175.157,34.562,156.401
C08692=1067.808,385.635,391.227,175.151,34.555,156.399
C08693=1067.800,385.388,391.267,175.147,34.547,156.397
C08694=1067.793,385.142,391.306,175.142,34.540,156.396
C08695=1067.787,384.895,391.346,175.138,34.533,156.394
C08696=1067.779,384.648,391.386,175.132,34.526,156.392
C08697=1067.772,384.402,391.426,175.128,34.519,156.391
C08698=1067.765,384.156,391.466,175.123,34.512,156.389
C08699=1067.758,383.909,391.506,175.118,34.504,156.388
C08700=1067.752,383.662,391.545,175.113,34.497,156.386
C08701=1067.744,383.415,391.585,175.109,34.490,156.384
C08702=1067.737,383.168,391.625,175.105,34.483,156.383
C08703=1067.730,382.922,391.665,175.099,34.476,156.381
C08704=1067.723,382.676,391.704,175.095,34.469,156.380
C08705=1067.716,382.428,391.744,175.090,34.462,156.378
C08706=1067.709,382.182,391.784,175.086,34.455,156.376
C08707=1067.702,381.936,391.823,175.080,34.448,156.375
C08708=1067.695,381.689,391.862,175.076,34.441,156.373
C08709=1067.688,381.442,391.902,175.071,34.434,156.372
C08710=1067.682,381.195,391.942,175.067,34.427,156.370
C08711=1067.675,380.948,391.981,175.062,34.420,156.369
C08712=1067.668,380.702,392.020,175.057,34.413,156.367
C08713=1067.660,380.455,392.060,175.053,34.406,156.366
C08714=1067.653,380.208,392.099,175.048,34.399,156.364
C08715=1067.646,379.962,392.138,175.043,34.392,156.363
C08716=1067.639,379.715,392.177,175.039,34.386,156.361
C08717=1067.632,379.468,392.217,175.034,34.379,156.360
C08718=1067.625,379.221,392.256,175.030,34.372,156.358
C08719=1067.618,378.974,392.295,175.025,34.365,156.356
C08720=1067.611,378.728,392.334,175.020,34.358,156.355
C08721=1067.604,378.481,392.373,175.016,34.351,156.354
C08722=1067.597,378.234,392.412,175.011,34.345,156.352
C08723=1067.590,377.987,392.451,175.007,34.338,156.351
C08724=1067.583,377.741,392.491,175.002,34.331,156.349
C08725=1067.576,377.494,392.529,174.998,34.324,156.348
C08726=1067.569,377.247,392.568,174.993,34.318,156.346
C08727=1067.562,377.000,392.607,174.988,34.311,156.345
C08728=1067.555,376.753,392.646,174.984,34.305,156.343
C08729=1067.549,376.507,392.685,174.980,34.298,156.342
C08730=1067.542,376.260,392.724,174.975,34.291,156.340
C08731=1067.535,376.013,392.763,174.971,34.284,156.339
C08732=1067.528,375.766,392.801,174.966,34.278,156.337
C08733=1067.521,375.519,392.841,174.962,34.271,156.336
C08734=1067.514,375.272,392.879,174.957,34.265,156.334
C08735=1067.507,375.025,392.918,174.952,34.258,156.333
C08736=1067.501,374.779,392.957,174.948,34.252,156.332
C08737=1067.493,374.532,392.995,174.944,34.245,156.330
C08738=1067.487,374.286,393.034,174.939,34.238,156.329
C08739=1067.480,374.039,393.073,174.935,34.232,156.327
C08740=1067.473,373.792,393.111,174.931,34.225,156.326
C08741=1067.466,373.551,393.149,174.926,34.219,156.324
C08742=1067.460,373.311,393.186,174.922,34.213,156.323
C08743=1067.453,373.072,393.224,174.918,34.206,156.322
C08744=1067.446,372.831,393.262,174.913,34.200,156.320
C08745=1067.440,372.591,393.299,174.909,34.194,156.319
C08746=1067.433,372.351,393.336,174.905,34.188,156.318
C08747=1067.426,372.111,393.373,174.900,34.181,156.316
C08748=1067.419,371.871,393.411,174.896,34.175,156.315
C08749=1067.413,371.624,393.449,174.892,34.169,156.314
C08750=1067.405,371.378,393.488,174.887,34.162,156.312
C08751=1067.399,371.130,393.526,174.883,34.156,156.311
C08752=1067.392,370.884,393.564,174.879,34.150,156.309
C08753=1067.385,370.637,393.602,174.875,34.143,156.308
C08754=1067.378,370.390,393.641,174.870,34.137,156.307
C08755=1067.371,370.143,393.678,174.866,34.131,156.305
C08756=1067.364,369.896,393.717,174.862,34.125,156.304
C08757=1067.358,369.649,393.755,174.857,34.118,156.303
C08758=1067.350,369.402,393.793,174.853,34.112,156.301
C08759=1067.344,369.155,393.831,174.849,34.106,156.300
C08760=1067.337,368.908,393.869,174.844,34.100,156.299
C08761=1067.330,368.661,393.907,174.840,34.093,156.297
C08762=1067.324,368.414,393.946,174.836,34.087,156.296
C08763=1067.317,368.167,393.983,174.832,34.081,156.294
C08764=1067.310,367.921,394.022,174.827,34.075,156.293
C08765=1067.303,367.674,394.059,174.823,34.068,156.292
C08766=1067.297,367.426,394.097,174.819,34.062,156.290
C08767=1067.289,367.179,394.135,174.814,34.056,156.289
C08768=1067.283,366.933,394.173,174.810,34.050,156.288
C08769=1067.276,366.686,394.211,174.806,34.044,156.286
C08770=1067.269,366.438,394.249,174.802,34.038,156.285
C08771=1067.263,366.191,394.287,174.797,34.031,156.284
C08772=1067.256,365.944,394.324,174.793,34.025,156.282
C08773=1067.250,365.697,394.362,174.790,34.019,156.281
C08774=1067.243,365.450,394.399,174.786,34.013,156.280
C08775=1067.237,365.203,394.438,174.781,34.007,156.279
C08776=1067.229,364.956,394.475,174.777,34.001,156.277
C08777=1067.223,364.709,394.513,174.773,33.995,156.276
C08778=1067.216,364.462,394.550,174.768,33.989,156.275
C08779=1067.209,364.215,394.588,174.764,33.983,156.273
C08780=1067.203,363.968,394.626,174.760,33.977,156.272
C08781=1067.196,363.721,394.663,174.756,33.971,156.271
C08782=1067.189,363.474,394.701,174.751,33.965,156.270
C08783=1067.183,363.227,394.738,174.747,33.959,156.268
C08784=1067.176,362.979,394.775,174.744,33.953,156.267
C08785=1067.169,362.733,394.812,174.740,33.947,156.266
C08786=1067.163,362.485,394.851,174.735,33.941,156.264
C08787=1067.155,362.238,394.888,174.731,33.935,156.263
C08788=1067.149,361.991,394.925,174.727,33.930,156.262
C08789=1067.142,361.744,394.962,174.723,33.923,156.261
C08790=1067.136,361.497,395.000,174.719,33.917,156.259
C08791=1067.129,361.250,395.037,174.714,33.912,156.258
C08792=1067.122,361.003,395.074,174.711,33.906,156.257
C08793=1067.115,360.756,395.111,174.707,33.900,156.256
C08794=1067.108,360.508,395.148,174.703,33.894,156.254
C08795=1067.102,360.262,395.186,174.698,33.888,156.253
C08796=1067.095,360.014,395.223,174.694,33.882,156.252
C08797=1067.089,359.783,395.258,174.691,33.877,156.251
C08798=1067.083,359.552,395.293,174.687,33.872,156.250
C08799=1067.076,359.320,395.327,174.683,33.866,156.249
C08800=1067.070,359.089,395.362,174.679,33.861,156.247
C08801=1067.064,358.858,395.396,174.675,33.855,156.246
C08802=1067.058,358.627,395.431,174.672,33.850,156.245
C08803=1067.052,358.395,395.465,174.668,33.844,156.244
C08804=1067.045,358.163,395.500,174.665,33.839,156.243
C08805=1067.038,357.916,395.537,174.660,33.834,156.242
C08806=1067.031,357.669,395.573,174.656,33.828,156.240
C08807=1067.025,357.422,395.611,174.652,33.822,156.239
C08808=1067.019,357.175,395.647,174.648,33.816,156.238
C08809=1067.012,356.927,395.684,174.645,33.811,156.237
C08810=1067.005,356.681,395.721,174.640,33.805,156.236
C08811=1066.998,356.433,395.758,174.636,33.800,156.235
C08812=1066.992,356.186,395.794,174.632,33.794,156.233
C08813=1066.985,355.939,395.831,174.628,33.788,156.232
C08814=1066.978,355.691,395.868,174.625,33.783,156.231
C08815=1066.972,355.445,395.905,174.620,33.777,156.230
C08816=1066.965,355.198,395.941,174.616,33.771,156.229
C08817=1066.958,354.950,395.978,174.612,33.765,156.227
C08818=1066.952,354.703,396.014,174.609,33.760,156.226
C08819=1066.946,354.456,396.051,174.605,33.754,156.225
C08820=1066.939,354.208,396.088,174.601,33.749,156.224
C08821=1066.933,353.961,396.124,174.596,33.743,156.223
C08822=1066.926,353.714,396.161,174.593,33.738,156.222
C08823=1066.919,353.466,396.197,174.589,33.732,156.220
C08824=1066.913,353.219,396.234,174.585,33.727,156.219
C08825=1066.907,352.972,396.270,174.581,33.721,156.218
C08826=1066.900,352.725,396.307,174.577,33.716,156.217
C08827=1066.893,352.477,396.344,174.573,33.710,156.216
C08828=1066.887,352.230,396.380,174.569,33.705,156.215
C08829=1066.880,351.984,396.416,174.566,33.699,156.213
C08830=1066.874,351.736,396.452,174.562,33.694,156.212
C08831=1066.867,351.488,396.488,174.558,33.688,156.211
C08832=1066.861,351.241,396.525,174.554,33.683,156.210
C08833=1066.854,350.994,396.561,174.550,33.677,156.209
C08834=1066.847,350.747,396.597,174.546,33.672,156.208
C08835=1066.841,350.499,396.633,174.542,33.666,156.207
C08836=1066.834,350.252,396.670,174.539,33.661,156.206
C08837=1066.827,350.005,396.705,174.535,33.655,156.204
C08838=1066.821,349.758,396.741,174.531,33.650,156.203
C08839=1066.815,349.511,396.778,174.527,33.645,156.202
C08840=1066.807,349.263,396.814,174.523,33.639,156.201
C08841=1066.801,349.015,396.850,174.519,33.634,156.200
C08842=1066.795,348.768,396.886,174.516,33.629,156.199
C08843=1066.789,348.521,396.922,174.512,33.623,156.198
C08844=1066.782,348.274,396.958,174.508,33.618,156.197
C08845=1066.776,348.026,396.993,174.504,33.612,156.195
C08846=1066.769,347.779,397.030,174.500,33.607,156.194
C08847=1066.762,347.531,397.065,174.496,33.602,156.193
C08848=1066.756,347.284,397.102,174.493,33.597,156.192
C08849=1066.749,347.037,397.137,174.489,33.591,156.191
C08850=1066.742,346.790,397.173,174.486,33.586,156.190
C08851=1066.736,346.542,397.209,174.482,33.581,156.189
C08852=1066.729,346.295,397.245,174.478,33.576,156.188
C08853=1066.724,346.065,397.278,174.474,33.570,156.187
C08854=1066.718,345.836,397.311,174.471,33.566,156.186
C08855=1066.711,345.607,397.344,174.467,33.560,156.185
C08856=1066.706,345.377,397.377,174.464,33.556,156.184
C08857=1066.700,345.148,397.411,174.461,33.551,156.183
C08858=1066.693,344.919,397.443,174.457,33.546,156.182
C08859=1066.688,344.689,397.477,174.454,33.541,156.181
C08860=1066.682,344.460,397.510,174.451,33.537,156.180
C08861=1066.676,344.234,397.542,174.446,33.532,156.179
C08862=1066.670,344.010,397.575,174.443,33.527,156.178
C08863=1066.664,343.785,397.607,174.440,33.522,156.177
C08864=1066.659,343.559,397.639,174.437,33.517,156.176
C08865=1066.652,343.312,397.674,174.433,33.512,156.175
C08866=1066.645,343.065,397.710,174.429,33.507,156.174
C08867=1066.639,342.818,397.746,174.426,33.502,156.173
C08868=1066.632,342.570,397.781,174.422,33.497,156.172
C08869=1066.625,342.323,397.816,174.419,33.492,156.171
C08870=1066.619,342.075,397.852,174.414,33.487,156.170
C08871=1066.612,341.828,397.887,174.411,33.482,156.169
C08872=1066.606,341.581,397.922,174.407,33.476,156.168
C08873=1066.600,341.333,397.958,174.403,33.471,156.166
C08874=1066.593,341.086,397.993,174.400,33.466,156.166
C08875=1066.586,340.838,398.028,174.396,33.461,156.164
C08876=1066.580,340.590,398.064,174.393,33.456,156.163
C08877=1066.573,340.343,398.099,174.389,33.451,156.162
C08878=1066.567,340.096,398.134,174.386,33.446,156.161
C08879=1066.561,339.847,398.169,174.381,33.440,156.160
C08880=1066.555,339.601,398.204,174.378,33.436,156.159
C08881=1066.548,339.353,398.239,174.374,33.430,156.158
C08882=1066.542,339.106,398.275,174.371,33.426,156.157
C08883=1066.535,338.858,398.310,174.367,33.420,156.156
C08884=1066.528,338.611,398.345,174.364,33.415,156.155
C08885=1066.522,338.363,398.379,174.360,33.410,156.154
C08886=1066.516,338.116,398.415,174.357,33.405,156.153
C08887=1066.510,337.869,398.450,174.353,33.400,156.152
C08888=1066.503,337.621,398.485,174.350,33.395,156.151
C08889=1066.496,337.373,398.519,174.346,33.390,156.150
C08890=1066.490,337.126,398.555,174.342,33.385,156.149
C08891=1066.484,336.878,398.590,174.338,33.380,156.148
C08892=1066.478,336.631,398.624,174.335,33.375,156.147
C08893=1066.471,336.384,398.659,174.331,33.370,156.146
C08894=1066.465,336.136,398.694,174.328,33.366,156.145
C08895=1066.458,335.888,398.729,174.324,33.360,156.144
C08896=1066.451,335.640,398.763,174.321,33.356,156.143
C08897=1066.445,335.394,398.798,174.317,33.350,156.142
C08898=1066.439,335.146,398.833,174.314,33.346,156.141
C08899=1066.432,334.898,398.868,174.310,33.341,156.140
C08900=1066.425,334.650,398.902,174.307,33.336,156.139
C08901=1066.419,334.404,398.937,174.304,33.331,156.138
C08902=1066.413,334.156,398.971,174.300,33.326,156.137
C08903=1066.406,333.908,399.006,174.296,33.322,156.136
C08904=1066.400,333.661,399.041,174.292,33.316,156.135
C08905=1066.393,333.414,399.076,174.289,33.312,156.134
C08906=1066.387,333.166,399.110,174.285,33.307,156.133
C08907=1066.381,332.918,399.144,174.282,33.301,156.132
C08908=1066.374,332.671,399.179,174.279,33.297,156.131
C08909=1066.369,332.427,399.213,174.275,33.292,156.130
C08910=1066.362,332.185,399.247,174.272,33.287,156.129
C08911=1066.356,331.942,399.281,174.268,33.282,156.128
C08912=1066.349,331.698,399.314,174.265,33.278,156.127
C08913=1066.344,331.455,399.349,174.262,33.273,156.126
C08914=1066.337,331.212,399.382,174.258,33.268,156.126
C08915=1066.331,330.969,399.416,174.255,33.264,156.125
C08916=1066.325,330.726,399.449,174.252,33.259,156.124
C08917=1066.318,330.479,399.484,174.248,33.254,156.123
C08918=1066.312,330.231,399.518,174.244,33.249,156.122
C08919=1066.305,329.984,399.552,174.241,33.245,156.121
C08920=1066.298,329.736,399.587,174.237,33.240,156.120
C08921=1066.293,329.489,399.621,174.234,33.235,156.119
C08922=1066.285,329.241,399.655,174.230,33.230,156.118
C08923=1066.279,328.993,399.689,174.227,33.226,156.117
C08924=1066.273,328.746,399.723,174.224,33.221,156.116
C08925=1066.266,328.498,399.757,174.220,33.216,156.115
C08926=1066.260,328.251,399.791,174.217,33.212,156.114
C08927=1066.253,328.003,399.825,174.213,33.207,156.113
C08928=1066.246,327.755,399.859,174.210,33.202,156.112
C08929=1066.241,327.508,399.893,174.207,33.198,156.111
C08930=1066.233,327.260,399.927,174.203,33.193,156.111
C08931=1066.227,327.013,399.961,174.200,33.188,156.110
C08932=1066.221,326.765,399.995,174.197,33.183,156.109
C08933=1066.215,326.517,400.028,174.193,33.179,156.108
C08934=1066.208,326.269,400.063,174.190,33.175,156.107
C08935=1066.202,326.022,400.096,174.187,33.170,156.106
C08936=1066.195,325.774,400.131,174.183,33.165,156.105
C08937=1066.189,325.527,400.165,174.180,33.160,156.104
C08938=1066.182,325.279,400.198,174.177,33.156,156.103
C08939=1066.177,325.031,400.232,174.172,33.151,156.102
C08940=1066.169,324.784,400.266,174.169,33.147,156.101
C08941=1066.163,324.536,400.300,174.166,33.142,156.100
C08942=1066.157,324.288,400.333,174.162,33.137,156.099
C08943=1066.151,324.041,400.367,174.159,33.132,156.099
C08944=1066.144,323.793,400.401,174.156,33.128,156.098
C08945=1066.138,323.545,400.434,174.152,33.123,156.097
C08946=1066.132,323.298,400.468,174.149,33.119,156.096
C08947=1066.125,323.050,400.502,174.146,33.114,156.095
C08948=1066.119,322.802,400.535,174.143,33.110,156.094
C08949=1066.112,322.555,400.569,174.139,33.105,156.093
C08950=1066.106,322.307,400.603,174.136,33.100,156.092
C08951=1066.100,322.060,400.636,174.133,33.095,156.091
C08952=1066.094,321.812,400.670,174.129,33.091,156.090
C08953=1066.087,321.564,400.703,174.126,33.086,156.089
C08954=1066.081,321.317,400.737,174.123,33.082,156.089
C08955=1066.074,321.069,400.770,174.120,33.077,156.088
C08956=1066.069,320.821,400.804,174.116,33.073,156.087
C08957=1066.062,320.574,400.837,174.113,33.068,156.086
C08958=1066.056,320.326,400.871,174.110,33.064,156.085
C08959=1066.050,320.078,400.904,174.107,33.059,156.084
C08960=1066.044,319.830,400.937,174.103,33.054,156.083
C08961=1066.037,319.583,400.971,174.100,33.050,156.082
C08962=1066.031,319.335,401.005,174.097,33.045,156.081
C08963=1066.025,319.088,401.038,174.094,33.040,156.080
C08964=1066.019,318.840,401.071,174.090,33.036,156.080
C08965=1066.013,318.605,401.102,174.087,33.031,156.079
C08966=1066.007,318.370,401.135,174.084,33.027,156.078
C08967=1066.002,318.135,401.166,174.081,33.023,156.077
C08968=1065.995,317.900,401.197,174.078,33.019,156.076
C08969=1065.990,317.666,401.229,174.075,33.015,156.075
C08970=1065.983,317.430,401.261,174.072,33.010,156.074
C08971=1065.978,317.196,401.292,174.069,33.006,156.074
C08972=1065.972,316.961,401.323,174.066,33.001,156.073
C08973=1065.966,316.713,401.357,174.063,32.997,156.072
C08974=1065.960,316.466,401.390,174.060,32.993,156.071
C08975=1065.954,316.218,401.423,174.056,32.988,156.070
C08976=1065.947,315.970,401.457,174.053,32.983,156.069
C08977=1065.942,315.722,401.490,174.050,32.979,156.068
C08978=1065.935,315.475,401.523,174.047,32.974,156.067
C08979=1065.929,315.228,401.556,174.044,32.970,156.067
C08980=1065.923,314.980,401.589,174.040,32.965,156.066
C08981=1065.917,314.732,401.622,174.037,32.961,156.065
C08982=1065.911,314.484,401.656,174.034,32.956,156.064
C08983=1065.905,314.237,401.688,174.031,32.952,156.063
C08984=1065.899,313.989,401.721,174.028,32.947,156.062
C08985=1065.892,313.741,401.754,174.024,32.943,156.061
C08986=1065.885,313.493,401.787,174.021,32.939,156.061
C08987=1065.879,313.246,401.820,174.018,32.934,156.060
C08988=1065.873,312.998,401.852,174.015,32.930,156.059
C08989=1065.867,312.750,401.885,174.012,32.925,156.058
C08990=1065.861,312.502,401.917,174.009,32.921,156.057
C08991=1065.854,312.254,401.950,174.005,32.917,156.056
C08992=1065.847,312.006,401.983,174.002,32.912,156.055
C08993=1065.841,311.759,402.016,173.999,32.908,156.055
C08994=1065.835,311.511,402.048,173.996,32.904,156.054
C08995=1065.828,311.264,402.081,173.993,32.899,156.053
C08996=1065.822,311.016,402.113,173.989,32.895,156.052
C08997=1065.816,310.768,402.145,173.986,32.890,156.051
C08998=1065.809,310.520,402.178,173.983,32.886,156.050
C08999=1065.803,310.273,402.211,173.980,32.882,156.050
C09000=1065.797,310.025,402.244,173.977,32.878,156.049
C09001=1065.791,309.777,402.276,173.974,32.873,156.048
C09002=1065.784,309.529,402.309,173.971,32.869,156.047
C09003=1065.777,309.281,402.341,173.967,32.864,156.046
C09004=1065.771,309.033,402.373,173.964,32.860,156.045
C09005=1065.764,308.786,402.406,173.961,32.856,156.045
C09006=1065.758,308.538,402.438,173.958,32.852,156.044
C09007=1065.752,308.290,402.470,173.955,32.848,156.043
C09008=1065.746,308.042,402.503,173.952,32.843,156.042
C09009=1065.740,307.794,402.535,173.949,32.839,156.041
C09010=1065.734,307.546,402.568,173.945,32.834,156.040
C09011=1065.727,307.299,402.600,173.942,32.830,156.040
C09012=1065.721,307.052,402.632,173.939,32.826,156.039
C09013=1065.715,306.804,402.664,173.936,32.822,156.038
C09014=1065.709,306.556,402.697,173.933,32.817,156.037
C09015=1065.703,306.308,402.729,173.930,32.813,156.036
C09016=1065.696,306.060,402.761,173.927,32.808,156.035
C09017=1065.690,305.813,402.793,173.924,32.804,156.035
C09018=1065.684,305.564,402.825,173.921,32.800,156.034
C09019=1065.677,305.317,402.858,173.917,32.796,156.033
C09020=1065.671,305.069,402.890,173.914,32.791,156.032
C09021=1065.666,304.836,402.920,173.911,32.787,156.031
C09022=1065.659,304.603,402.951,173.909,32.783,156.031
C09023=1065.654,304.370,402.981,173.906,32.779,156.030
C09024=1065.648,304.137,403.011,173.903,32.775,156.029
C09025=1065.642,303.904,403.041,173.900,32.771,156.028
C09026=1065.636,303.671,403.071,173.897,32.767,156.028
C09027=1065.630,303.438,403.101,173.894,32.763,156.027
C09028=1065.625,303.205,403.132,173.891,32.759,156.026
C09029=1065.618,302.957,403.164,173.888,32.754,156.025
C09030=1065.613,302.710,403.195,173.885,32.750,156.024
C09031=1065.607,302.461,403.227,173.882,32.746,156.024
C09032=1065.600,302.214,403.260,173.879,32.742,156.023
C09033=1065.594,301.966,403.291,173.876,32.737,156.022
C09034=1065.588,301.718,403.324,173.873,32.733,156.021
C09035=1065.582,301.470,403.355,173.870,32.729,156.020
C09036=1065.576,301.223,403.388,173.867,32.725,156.019
C09037=1065.569,300.975,403.419,173.865,32.721,156.019
C09038=1065.563,300.726,403.451,173.862,32.716,156.018
C09039=1065.558,300.479,403.483,173.859,32.712,156.017
C09040=1065.552,300.231,403.515,173.856,32.708,156.016
C09041=1065.545,299.983,403.546,173.853,32.704,156.015
C09042=1065.540,299.735,403.578,173.850,32.699,156.014
C09043=1065.534,299.488,403.611,173.847,32.695,156.014
C09044=1065.527,299.240,403.642,173.844,32.690,156.013
C09045=1065.521,298.992,403.674,173.841,32.686,156.012
C09046=1065.515,298.744,403.706,173.838,32.682,156.011
C09047=1065.509,298.496,403.738,173.835,32.678,156.010
C09048=1065.503,298.249,403.769,173.832,32.673,156.010
C09049=1065.497,298.001,403.801,173.829,32.669,156.009
C09050=1065.491,297.752,403.833,173.826,32.665,156.008
C09051=1065.485,297.505,403.864,173.823,32.661,156.007
C09052=1065.479,297.257,403.896,173.820,32.656,156.006
C09053=1065.473,297.009,403.928,173.817,32.652,156.006
C09054=1065.467,296.761,403.959,173.814,32.648,156.005
C09055=1065.461,296.513,403.990,173.811,32.644,156.004
C09056=1065.455,296.265,404.022,173.808,32.639,156.003
C09057=1065.449,296.018,404.053,173.805,32.636,156.002
C09058=1065.443,295.769,404.085,173.802,32.631,156.002
C09059=1065.436,295.521,404.117,173.799,32.627,156.001
C09060=1065.431,295.273,404.148,173.796,32.623,156.000
C09061=1065.424,295.025,404.179,173.794,32.619,155.999
C09062=1065.417,294.777,404.210,173.791,32.614,155.998
C09063=1065.412,294.530,404.242,173.788,32.611,155.998
C09064=1065.406,294.281,404.273,173.785,32.606,155.997
C09065=1065.399,294.034,404.304,173.782,32.602,155.996
C09066=1065.393,293.786,404.336,173.779,32.598,155.995
C09067=1065.387,293.538,404.367,173.776,32.594,155.995
C09068=1065.380,293.290,404.398,173.773,32.590,155.994
C09069=1065.375,293.042,404.430,173.770,32.586,155.993
C09070=1065.368,292.794,404.461,173.767,32.581,155.992
C09071=1065.362,292.546,404.491,173.764,32.577,155.991
C09072=1065.356,292.298,404.523,173.761,32.573,155.991
C09073=1065.350,292.050,404.554,173.758,32.569,155.990
C09074=1065.344,291.802,404.585,173.755,32.565,155.989
C09075=1065.337,291.554,404.616,173.752,32.561,155.988
C09076=1065.331,291.307,404.647,173.750,32.557,155.988
C09077=1065.326,291.081,404.675,173.747,32.553,155.987
C09078=1065.320,290.855,404.704,173.744,32.549,155.986
C09079=1065.315,290.630,404.732,173.742,32.546,155.985
C09080=1065.309,290.405,404.761,173.740,32.542,155.985
C09081=1065.304,290.179,404.789,173.737,32.538,155.984
C09082=1065.298,289.954,404.817,173.735,32.534,155.983
C09083=1065.292,289.729,404.845,173.732,32.530,155.983
C09084=1065.287,289.503,404.873,173.729,32.527,155.982
C09085=1065.280,289.255,404.904,173.726,32.522,155.981
C09086=1065.275,289.006,404.935,173.723,32.519,155.980
C09087=1065.269,288.759,404.966,173.721,32.514,155.980
C09088=1065.262,288.510,404.997,173.718,32.510,155.979
C09089=1065.256,288.263,405.027,173.715,32.506,155.978
C09090=1065.250,288.015,405.059,173.712,32.502,155.977
C09091=1065.244,287.767,405.089,173.709,32.498,155.977
C09092=1065.237,287.518,405.120,173.706,32.494,155.976
C09093=1065.232,287.271,405.150,173.703,32.490,155.975
C09094=1065.225,287.023,405.182,173.700,32.486,155.974
C09095=1065.219,286.775,405.212,173.698,32.482,155.974
C09096=1065.213,286.526,405.243,173.695,32.478,155.973
C09097=1065.207,286.278,405.273,173.693,32.473,155.972
C09098=1065.201,286.031,405.304,173.690,32.470,155.971
C09099=1065.194,285.783,405.335,173.687,32.465,155.970
C09100=1065.188,285.535,405.365,173.684,32.462,155.970
C09101=1065.182,285.286,405.396,173.681,32.457,155.969
C09102=1065.176,285.039,405.426,173.678,32.453,155.968
C09103=1065.170,284.791,405.458,173.675,32.449,155.968
C09104=1065.164,284.543,405.488,173.672,32.445,155.967
C09105=1065.158,284.295,405.518,173.670,32.441,155.966
